    3:
	   HMI_AxisView[47].MoveReal:=FALSE;
       DO_[31,6].ON:=TRUE;
	   iAutoCut:=4;	
    4:
       tonAutoCut(IN:= TRUE, PT:= T#2S, Q=> , ET=> ); 
	   IF tonAutoCut.Q THEN 
	       tonAutoCut(IN:= FALSE, PT:= T#2S, Q=> , ET=> ); 
           iAutoCut:=5;	   
	   END_IF	
	   
    5: DO_[31,6].ON:=FALSE;
	   iAutoCut:=6;	
    6: 	  
       tonAutoCut(IN:= TRUE, PT:= T#3S, Q=> , ET=> ); 
	   IF tonAutoCut.Q THEN 
	       tonAutoCut(IN:= FALSE, PT:= T#3S, Q=> , ET=> ); 
           iAutoCut:=7;	   
	   END_IF	
    7: 
 	   IF icutcnt> HMI_cutCnt THEN
		  iAutoCut:=8; 
	   ELSE 
	      iAutoCut:=0; 
	   END_IF
	8:   
       HMI_AxisView[46].MoveReal:=TRUE;
	   iAutoCut:=9;	  
 
	9:
       tonAutoCut(IN:= TRUE, PT:= T#2S, Q=> , ET=> ); 
	   IF tonAutoCut.Q THEN 
	       tonAutoCut(IN:= FALSE, PT:= T#2S, Q=> , ET=> ); 
           iAutoCut:=10;	   
	   END_IF	
	   
	10:
	   icutcnt:=0;
       HMI_AxisView[46].MoveReal:=FALSE;
	   iAutoCut:=0;		   
	   
END_CASE


tonCounterAirOpen(IN:= glb_bCounterAirValve_UN01 , PT:= T#3S, Q=> , ET=> );
IF tonCounterAirOpen.Q THEN
   glb_bPackAirValve_UN01:=TRUE;
END_IF


IF HMI_DisableCntAlarmAll THEN
	FOR  i:=1 TO 40 DO
		HMI_SkipCntAlarm[i]:=TRUE;
	END_FOR
END_IF

IF HMI_EnbaleCntAlarmAll THEN
	FOR  i:=1 TO 40 DO
		HMI_SkipCntAlarm[i]:=FALSE;
	END_FOR	
END_IF

IF HMI_DisableCntAlarmAll2 THEN
	FOR  i:=1 TO 40 DO
		HMI_CntCheck[i]:=TRUE;
	END_FOR
END_IF

IF HMI_EnbaleCntAlarmAll2 THEN
	FOR  i:=1 TO 40 DO
		HMI_CntCheck[i]:=FALSE;
	END_FOR	
END_IF
END_ACTION

ACTION SR90_SafetyReset:
CASE iSafetyResetSeq OF
	0: IF glb_bSafetyReset THEN
		  iSafetyResetSeq:=10;
	   END_IF
	10: 	
		IF glb_arSafeRelayNo_UN01[1] OR tonSafetyReset.Q  THEN
		    iSafetyResetSeq:=20;
		END_IF
	20:	
		FOR i:=1 TO 64 DO
		    arRealAxisAdmin[i].i.Reset:= TRUE ;
			iSafetyResetSeq:=30;
		END_FOR		
	30:
	    IF tonSafetyReset.Q THEN
		   FOR i:=1 TO 64 DO
		       arRealAxisAdmin[i].i.Reset:= FALSE ;	
	       END_FOR	
		   glb_bSafetyreset:=FALSE;
		   iSafetyResetSeq:=0;
		END_IF
	
END_CASE

tonSafetyReset(IN:=glb_bSafetyreset , PT:=T#3S , Q=> , ET=> );

	
IF glb_arSafeRelayNo_UN01[1] THEN
	glb_bAllSafetyOk:=TRUE;
	ELSE 
	glb_bAllSafetyOk:=FALSE;
END_IF
END_ACTION

ACTION SR91_OEE:
HMI_OEEView.Active:=TRUE;
IF HMI_OEEView.Active THEN
   IF rtGoodCount.Q THEN	
      HMI_OEEView.GoodCount:= HMI_OEEView.GoodCount+7;	
   END_IF 
   IF rtNoGoodCount.Q THEN
	  HMI_OEEView.NoGoodCount:= HMI_OEEView.NoGoodCount+7;
   END_IF
  
END_IF

rtGoodCount(CLK:= glb_digoodFlag_UN01.11, Q=> );
rtNoGoodCount(CLK:= glb_diNogoodFlag_UN01.11 , Q=> );

IF HMI_OEEView.Reset THEN
   HMI_OEEView.GoodCount:=0;
   HMI_OEEView.NoGoodCount:=0;	
END_IF


HMI_OEEView.DesignSpeed:= 7.5;
HMI_OEEView.Performance:=HMI_OEEView.AverageSpeed/HMI_OEEView.DesignSpeed*100;


aoiActiveTotalTime(
	bEnable:= HMI_OEEView.Active, 
	bReset:= HMI_OEEView.Reset, 
	diSecond=> , 
	diMinute=> , 
	diHour=> , 
	diTotalSecond=> , 
	diTotalMinute=> HMI_OEEView.PlannedTime, 
	diTotalHour=> );

aoiWorkTotalTime(
	bEnable:= HMI_OEEView.Active AND Ref_MachineStateModel.Sts_Execute, 
	bReset:= HMI_OEEView.Reset, 
	diSecond=> , 
	diMinute=> , 
	diHour=> , 
	diTotalSecond=> , 
	diTotalMinute=> HMI_OEEView.UsableTime, 
	diTotalHour=> );

aoi10MinuteTime(
	bEnable:= bEn10Minute OR TRUE, 
	bReset:= bReset10Minute, 
	diSecond=> , 
	diMinute=> , 
	diHour=> , 
	diTotalSecond=> , 
	diTotalMinute=> , 
	diTotalHour=> );
	

HMI_OEEView.AverageSpeed:=DINT_TO_REAL(glb_TransferCnt)*7/DINT_TO_REAL(aoiWorkTotalTime.diTotalMinute);

	
IF	aoiActiveTotalTime.diTotalMinute>0 THEN
    HMI_OEEView.Usability:= DINT_TO_REAL(aoiWorkTotalTime.diTotalMinute)/DINT_TO_REAL(aoiActiveTotalTime.diTotalMinute)*100;
ELSE
    HMI_OEEView.Usability:= 0;
END_IF	

IF (HMI_OEEView.NoGoodCount+HMI_OEEView.GoodCount)> 0 THEN
    HMI_OEEView.Quality:=DINT_TO_REAL(HMI_OEEView.GoodCount)/(DINT_TO_REAL(HMI_OEEView.NoGoodCount)+DINT_TO_REAL(HMI_OEEView.GoodCount))*100;
ELSE
	HMI_OEEView.Quality:=0;
END_IF

HMI_OEEView.OEE:=(HMI_OEEView.Quality/100*HMI_OEEView.Usability/100*HMI_OEEView.Performance/100)*100;
END_ACTION

ACTION SR99_FaultClear:
CASE iFaultClearSeq OF
	0: 
		IF bClearAllFault THEN
		   iFaultClearSeq:=10;
		END_IF
	   
	10: 	
	//    IF NOT glb_bAirFeedback_UN01[2] THEN
	//		glb_bCounterAirValve_UN01:=FALSE;
	//	END_IF
	
	//	IF NOT glb_bAirFeedback_UN01[1] THEN
	//		glb_bPackAirValve_UN01:=FALSE;
	//	END_IF
		
		glb_MembraneAlarm:=FALSE;
		FOR i:=1 TO 50 DO
			IF arRealAxisAdmin[i].o.Error  THEN
			   arRealAxisAdmin[i].i.Reset:= TRUE ;
			END_IF
			IF arVirtualAxisAdmin[i].o.Error THEN
			   arVirtualAxisAdmin[i].i.Reset:= TRUE ;
			END_IF
		END_FOR
	
		FOR j:=1 TO 40 DO
			IF arDropCylinder[j].o.Error THEN
		       arDropCylinder[j].i.Reset:=TRUE;
			END_IF
			IF arCounters[j].Error THEN
			   arCounters[j].Clear:=TRUE;
			END_IF
		END_FOR
	    FOR j:=1 TO 50 DO
 			IF arPackCylinder[j].o.Error THEN
		       arPackCylinder[j].i.Reset:=TRUE;
			END_IF
			IF arPackVacuum[j].o.Error THEN
		       arPackVacuum[j].i.Reset:=TRUE;
			END_IF  
		END_FOR		
		
		FOR j:=1 TO 8 DO
			arHeat_AOI[j].Reset:=TRUE;
		END_FOR
        arDropBufferCyclinder[1].i.Reset:=TRUE;
		arDropBufferCyclinder[2].i.Reset:=TRUE;
	    iFaultClearSeq:=20;

	20:
		HMI_StopEvent[5].ID[20]:=FALSE;
		HMI_StopEvent[5].ID[21]:=FALSE;
		HMI_StopEvent[5].ID[22]:=FALSE;
		HMI_StopEvent[5].ID[23]:=FALSE;
		HMI_StopEvent[5].ID[24]:=FALSE;
		HMI_StopEvent[5].ID[25]:=FALSE;
		HMI_StopEvent[5].ID[26]:=FALSE;
	
	   IF  tonFaultClear.Q THEN 
			FOR i:=1 TO 50 DO
				 arRealAxisAdmin[i].i.Reset:= FALSE ;
				 arVirtualAxisAdmin[i].i.Reset:= FALSE ;
			END_FOR
			FOR j:=1 TO 40 DO
				arDropCylinder[j].i.Reset:=FALSE;
			    arCounters[j].Clear:=FALSE;				
			END_FOR
			FOR j:=1 TO 50 DO
				arPackCylinder[j].i.Reset:=FALSE;
				arPackVacuum[j].i.Reset:=FALSE;
			END_FOR			
			
			FOR j:=1 TO 8 DO
				arHeat_AOI[j].Reset:=FALSE;
			END_FOR
		    HMI_PrinterFault:=FALSE;
			
		    HMI_StopEvent[0].ID[6]:=FALSE;
		    HMI_StopEvent[0].ID[7]:=FALSE;
			
		//	glb_bPackAirValve_UN01:=TRUE;
		//	glb_bCounterAirValve_UN01:=TRUE;
		
		    arDropBufferCyclinder[1].i.Reset:=FALSE;
		    arDropBufferCyclinder[2].i.Reset:=FALSE;
		
			HMI_AlarmMute:=FALSE;
			bClearAllFault:=FALSE;
			iFaultClearSeq:=0;
       END_IF
	   
END_CASE

tonFaultClear(IN:=bClearAllFault , PT:=T#500MS , Q=> , ET=> );
END_ACTION

ACTION UP01_PackML:
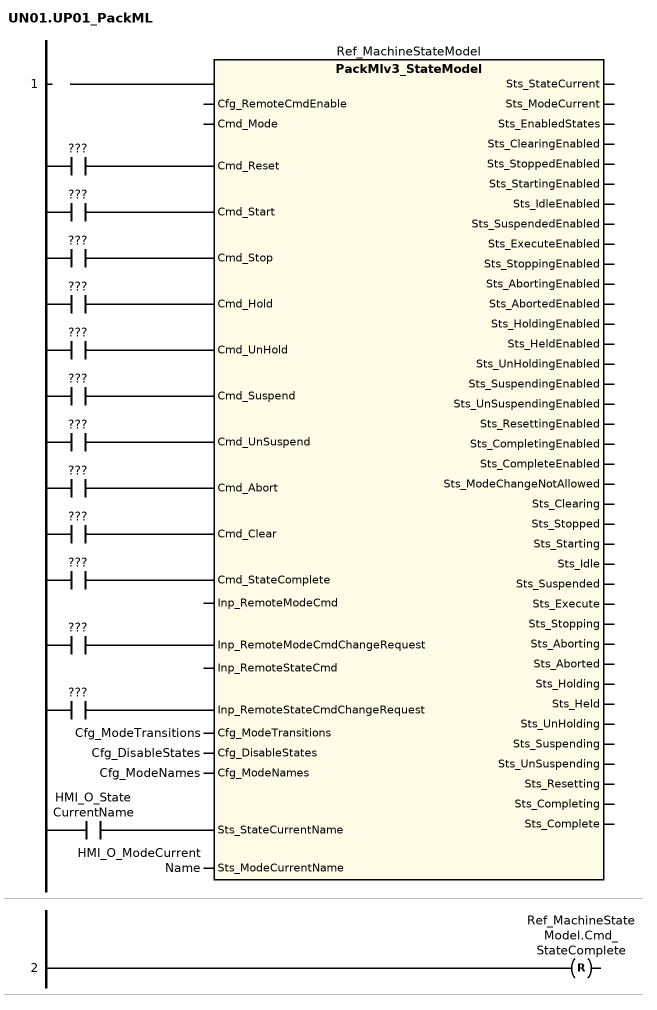
// NETWORK 1
Ref_MachineStateModel(
    Cfg_ModeTransitions := Cfg_ModeTransitions,
    Cfg_DisableStates := Cfg_DisableStates,
    Cfg_ModeNames := Cfg_ModeNames,
    Sts_StateCurrentName := HMI_O_StateCurrentName,
    Sts_ModeCurrentName := HMI_O_ModeCurrentName); // PackMlv3_StateModel

// NETWORK 2
Ref_MachineStateModel.Cmd_StateComplete R= TRUE;
END_ACTION

ACTION UP02_StateComplete:
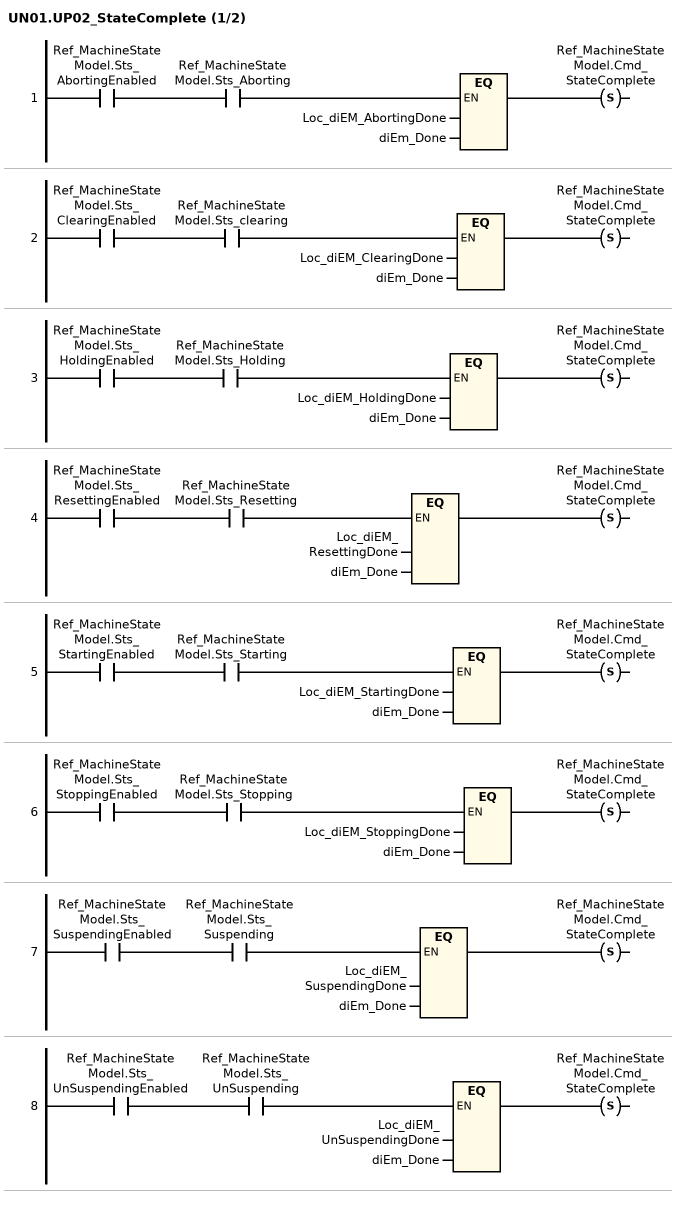
// NETWORK 1
Ref_MachineStateModel.Cmd_StateComplete S= Ref_MachineStateModel.Sts_AbortingEnabled AND Ref_MachineStateModel.Sts_Aborting AND Loc_diEM_AbortingDone = diEm_Done;

// NETWORK 2
Ref_MachineStateModel.Cmd_StateComplete S= Ref_MachineStateModel.Sts_ClearingEnabled AND Ref_MachineStateModel.Sts_clearing AND Loc_diEM_ClearingDone = diEm_Done;

// NETWORK 3
Ref_MachineStateModel.Cmd_StateComplete S= Ref_MachineStateModel.Sts_HoldingEnabled AND Ref_MachineStateModel.Sts_Holding AND Loc_diEM_HoldingDone = diEm_Done;

// NETWORK 4
Ref_MachineStateModel.Cmd_StateComplete S= Ref_MachineStateModel.Sts_ResettingEnabled AND Ref_MachineStateModel.Sts_Resetting AND Loc_diEM_ResettingDone = diEm_Done;

// NETWORK 5
Ref_MachineStateModel.Cmd_StateComplete S= Ref_MachineStateModel.Sts_StartingEnabled AND Ref_MachineStateModel.Sts_Starting AND Loc_diEM_StartingDone = diEm_Done;

// NETWORK 6
Ref_MachineStateModel.Cmd_StateComplete S= Ref_MachineStateModel.Sts_StoppingEnabled AND Ref_MachineStateModel.Sts_Stopping AND Loc_diEM_StoppingDone = diEm_Done;

// NETWORK 7
Ref_MachineStateModel.Cmd_StateComplete S= Ref_MachineStateModel.Sts_SuspendingEnabled AND Ref_MachineStateModel.Sts_Suspending AND Loc_diEM_SuspendingDone = diEm_Done;

// NETWORK 8
Ref_MachineStateModel.Cmd_StateComplete S= Ref_MachineStateModel.Sts_UnSuspendingEnabled AND Ref_MachineStateModel.Sts_UnSuspending AND Loc_diEM_UnSuspendingDone = diEm_Done;

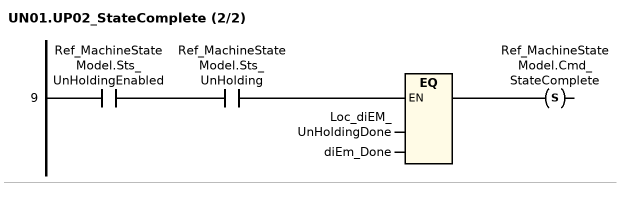
// NETWORK 9
Ref_MachineStateModel.Cmd_StateComplete S= Ref_MachineStateModel.Sts_UnHoldingEnabled AND Ref_MachineStateModel.Sts_UnHolding AND Loc_diEM_UnHoldingDone = diEm_Done;
END_ACTION

END_PROGRAM

// ---- Add-On-Instructions/PackMlv3_StateModel.TcPOU
FUNCTION_BLOCK PackMlv3_StateModel
VAR_INPUT
	Cfg_RemoteCmdEnable: BOOL;
	Cmd_Mode: DINT;
	Cmd_Reset: BOOL;
	Cmd_Start: BOOL;
	Cmd_Stop: BOOL;
	Cmd_Hold: BOOL;
	Cmd_UnHold: BOOL;
	Cmd_Suspend: BOOL;
	Cmd_UnSuspend: BOOL;
	Cmd_Abort: BOOL;
	Cmd_Clear: BOOL;
	Cmd_StateComplete: BOOL;
	Inp_RemoteModeCmd: DINT;
	Inp_RemoteModeCmdChangeRequest: BOOL;
	Inp_RemoteStateCmd: DINT;
	Inp_RemoteStateCmdChangeRequest: BOOL;
END_VAR
VAR_OUTPUT
	Sts_StateCurrent: DINT;
	Sts_ModeCurrent: DINT;
	Sts_EnabledStates: DINT;
	Sts_ClearingEnabled: BOOL;
	Sts_StoppedEnabled: BOOL;
	Sts_StartingEnabled: BOOL;
	Sts_IdleEnabled: BOOL;
	Sts_SuspendedEnabled: BOOL;
	Sts_ExecuteEnabled: BOOL;
	Sts_StoppingEnabled: BOOL;
	Sts_AbortingEnabled: BOOL;
	Sts_AbortedEnabled: BOOL;
	Sts_HoldingEnabled: BOOL;
	Sts_HeldEnabled: BOOL;
	Sts_UnHoldingEnabled: BOOL;
	Sts_SuspendingEnabled: BOOL;
	Sts_UnSuspendingEnabled: BOOL;
	Sts_ResettingEnabled: BOOL;
	Sts_CompletingEnabled: BOOL;
	Sts_CompleteEnabled: BOOL;
	Sts_ModeChangeNotAllowed: BOOL;
	Sts_Clearing: BOOL;
	Sts_Stopped: BOOL;
	Sts_Starting: BOOL;
	Sts_Idle: BOOL;
	Sts_Suspended: BOOL;
	Sts_Execute: BOOL;
	Sts_Stopping: BOOL;
	Sts_Aborting: BOOL;
	Sts_Aborted: BOOL;
	Sts_Holding: BOOL;
	Sts_Held: BOOL;
	Sts_UnHolding: BOOL;
	Sts_Suspending: BOOL;
	Sts_UnSuspending: BOOL;
	Sts_Resetting: BOOL;
	Sts_Completing: BOOL;
	Sts_Complete: BOOL;
END_VAR
VAR_IN_OUT
	Cfg_ModeTransitions: ARRAY[0..31] OF DINT;
	Cfg_DisableStates: ARRAY[0..31] OF DINT;
	Cfg_ModeNames: ARRAY[0..31] OF STRING;
	Sts_StateCurrentName: STRING(255);	
	Sts_ModeCurrentName: STRING(255);	
END_VAR
VAR
	RemoteCmdChangeRequested: BOOL;
	ResetRemoteCmd: BOOL;
	StartRemoteCmd: BOOL;
	StopRemoteCmd: BOOL;
	HoldRemoteCmd: BOOL;
	UnholdRemoteCmd: BOOL;
	SuspendRemoteCmd: BOOL;
	UnSuspendRemoteCmd: BOOL;
	AbortRemoteCmd: BOOL;
	ClearRemoteCmd: BOOL;
	Cfg_DisableStatesCopy: DINT;
	StateComplete: BOOL;
	LocalClearing: BOOL;
	LocalStopped: BOOL;
	LocalStarting: BOOL;
	LocalExecute: BOOL;
	LocalCompleting: BOOL;
	LocalStopping: BOOL;
	LocalAborting: BOOL;
	LocalAborted: BOOL;
	LocalHolding: BOOL;
	LocalHeld: BOOL;
	LocalUnHolding: BOOL;
	LocalSuspending: BOOL;
	LocalSuspended: BOOL;
	LocalUnSuspending: BOOL;
	LocalResetting: BOOL;
	LocalIdle: BOOL;
	LocalComplete: BOOL;
	END_IFIF: INT;
	FS: BOOL;
END_VAR
VAR // added by the converter: edge detectors and wires of the graphical bodies
    _w1, _w2, _w3, _w4, _w5, _w6, _w7, _w8, _w9, _w10, _w11, _w12, _w13, _w14, _w15, _w16, _w17, _w18, _w19, _w20, _w21, _w22, _w23, _w24, _w25, _w26, _w27, _w28, _w29, _w30, _w31, _w32, _w33, _w34, _w35, _w36, _w37, _w38, _w39, _w40, _w41, _w42, _w43, _w44, _w45, _w46, _w47, _w48, _w49, _w50, _w51, _w52, _w53, _w54, _w55, _w56 : BOOL;
END_VAR


IF NOT FS THEN
	Sts_ModeCurrent:=1;
	Cmd_Mode:=1;
	StS_StateCurrent:=2;
    LocalClearing:=FALSE;
	LocalStopped:=TRUE;
	LocalStarting:=FALSE;
	LocalExecute:=FALSE;
	LocalCompleting:=FALSE;
	LocalStopping:=FALSE;
	LocalAborting:=FALSE;
	LocalAborted:=FALSE;
	LocalHolding:=FALSE;
	LocalHeld:=FALSE;
	LocalUnHolding:=FALSE;
	LocalSuspending:=FALSE;
	LocalSuspended:=FALSE;
	LocalUnSuspending:=FALSE;
	LocalResetting:=FALSE;
	LocalIdle:=FALSE;
	LocalComplete:=FALSE;
	FS:=TRUE;
END_IF
ACT();

IF Sts_StateCurrent=0 THEN
	IF RemoteCmdchangerequested AND inp_remoteModeCmd<>0 AND Inp_RemoteModeCmd>1 AND Inp_RemoteModeCmd<32 
	 AND Cfg_ModeTransitions[Sts_ModeCurrent].0 AND Cfg_ModeTransitions[Inp_RemoteModeCmd].0 THEN
		Sts_ModeCurrent:=Inp_RemoteModeCmd;
		Cmd_Mode:=Sts_ModeCurrent;
	END_IF
	IF Cmd_Mode<>Sts_ModeCurrent AND Cmd_Mode>1 AND Cmd_Mode<32 
	 AND Cfg_ModeTransitions[Sts_ModeCurrent].0 AND Cfg_ModeTransitions[Cmd_Mode].0 THEN	
		Sts_ModeCurrent:=Cmd_Mode;
	END_IF
	
END_IF
IF Sts_StateCurrent=1 THEN
	IF RemoteCmdchangerequested AND inp_remoteModeCmd<>0 AND Inp_RemoteModeCmd>1 AND Inp_RemoteModeCmd<32 
	 AND Cfg_ModeTransitions[Sts_ModeCurrent].1 AND Cfg_ModeTransitions[Inp_RemoteModeCmd].1 THEN
		Sts_ModeCurrent:=Inp_RemoteModeCmd;
		Cmd_Mode:=Sts_ModeCurrent;
	END_IF
	IF Cmd_Mode<>Sts_ModeCurrent AND Cmd_Mode>1 AND Cmd_Mode<32 
	 AND Cfg_ModeTransitions[Sts_ModeCurrent].1 AND Cfg_ModeTransitions[Cmd_Mode].1 THEN	
		Sts_ModeCurrent:=Cmd_Mode;
	END_IF
END_IF
IF Sts_StateCurrent=2 THEN
	IF RemoteCmdchangerequested AND inp_remoteModeCmd<>0 AND Inp_RemoteModeCmd>1 AND Inp_RemoteModeCmd<32 
	 AND Cfg_ModeTransitions[Sts_ModeCurrent].2 AND Cfg_ModeTransitions[Inp_RemoteModeCmd].2 THEN
		Sts_ModeCurrent:=Inp_RemoteModeCmd;
		Cmd_Mode:=Sts_ModeCurrent;
	END_IF
	IF Cmd_Mode<>Sts_ModeCurrent AND Cmd_Mode>1 AND Cmd_Mode<32 
	 AND Cfg_ModeTransitions[Sts_ModeCurrent].2 AND Cfg_ModeTransitions[Cmd_Mode].2 THEN	
		Sts_ModeCurrent:=Cmd_Mode;
	END_IF
END_IF
IF Sts_StateCurrent=3 THEN
	IF RemoteCmdchangerequested AND inp_remoteModeCmd<>0 AND Inp_RemoteModeCmd>1 AND Inp_RemoteModeCmd<32 
	 AND Cfg_ModeTransitions[Sts_ModeCurrent].3 AND Cfg_ModeTransitions[Inp_RemoteModeCmd].3 THEN
		Sts_ModeCurrent:=Inp_RemoteModeCmd;
		Cmd_Mode:=Sts_ModeCurrent;
	END_IF
	IF Cmd_Mode<>Sts_ModeCurrent AND Cmd_Mode>1 AND Cmd_Mode<32 
	 AND Cfg_ModeTransitions[Sts_ModeCurrent].3 AND Cfg_ModeTransitions[Cmd_Mode].3 THEN	
		Sts_ModeCurrent:=Cmd_Mode;
	END_IF
END_IF
IF Sts_StateCurrent=4 THEN
	IF RemoteCmdchangerequested AND inp_remoteModeCmd<>0 AND Inp_RemoteModeCmd>1 AND Inp_RemoteModeCmd<32 
	 AND Cfg_ModeTransitions[Sts_ModeCurrent].4 AND Cfg_ModeTransitions[Inp_RemoteModeCmd].4 THEN
		Sts_ModeCurrent:=Inp_RemoteModeCmd;
		Cmd_Mode:=Sts_ModeCurrent;
	END_IF
	IF Cmd_Mode<>Sts_ModeCurrent AND Cmd_Mode>1 AND Cmd_Mode<32 
	 AND Cfg_ModeTransitions[Sts_ModeCurrent].4 AND Cfg_ModeTransitions[Cmd_Mode].4 THEN	
		Sts_ModeCurrent:=Cmd_Mode;
	END_IF
END_IF
IF Sts_StateCurrent=5 THEN
	IF RemoteCmdchangerequested AND inp_remoteModeCmd<>0 AND Inp_RemoteModeCmd>1 AND Inp_RemoteModeCmd<32 
	 AND Cfg_ModeTransitions[Sts_ModeCurrent].5 AND Cfg_ModeTransitions[Inp_RemoteModeCmd].5 THEN
		Sts_ModeCurrent:=Inp_RemoteModeCmd;
		Cmd_Mode:=Sts_ModeCurrent;
	END_IF
	IF Cmd_Mode<>Sts_ModeCurrent AND Cmd_Mode>1 AND Cmd_Mode<32 
	 AND Cfg_ModeTransitions[Sts_ModeCurrent].5 AND Cfg_ModeTransitions[Cmd_Mode].5 THEN	
		Sts_ModeCurrent:=Cmd_Mode;
	END_IF
END_IF
IF Sts_StateCurrent=6 THEN
	IF RemoteCmdchangerequested AND inp_remoteModeCmd<>0 AND Inp_RemoteModeCmd>1 AND Inp_RemoteModeCmd<32 
	 AND Cfg_ModeTransitions[Sts_ModeCurrent].6 AND Cfg_ModeTransitions[Inp_RemoteModeCmd].6 THEN
		Sts_ModeCurrent:=Inp_RemoteModeCmd;
		Cmd_Mode:=Sts_ModeCurrent;
	END_IF
	IF Cmd_Mode<>Sts_ModeCurrent AND Cmd_Mode>1 AND Cmd_Mode<32 
	 AND Cfg_ModeTransitions[Sts_ModeCurrent].6 AND Cfg_ModeTransitions[Cmd_Mode].6 THEN	
		Sts_ModeCurrent:=Cmd_Mode;
	END_IF
END_IF
IF Sts_StateCurrent=7 THEN
	IF RemoteCmdchangerequested AND inp_remoteModeCmd<>0 AND Inp_RemoteModeCmd>1 AND Inp_RemoteModeCmd<32 
	 AND Cfg_ModeTransitions[Sts_ModeCurrent].7 AND Cfg_ModeTransitions[Inp_RemoteModeCmd].7 THEN
		Sts_ModeCurrent:=Inp_RemoteModeCmd;
		Cmd_Mode:=Sts_ModeCurrent;
	END_IF
	IF Cmd_Mode<>Sts_ModeCurrent AND Cmd_Mode>1 AND Cmd_Mode<32 
	 AND Cfg_ModeTransitions[Sts_ModeCurrent].7 AND Cfg_ModeTransitions[Cmd_Mode].7 THEN	
		Sts_ModeCurrent:=Cmd_Mode;
	END_IF
END_IF
IF Sts_StateCurrent=8 THEN
	IF RemoteCmdchangerequested AND inp_remoteModeCmd<>0 AND Inp_RemoteModeCmd>1 AND Inp_RemoteModeCmd<32 
	 AND Cfg_ModeTransitions[Sts_ModeCurrent].8 AND Cfg_ModeTransitions[Inp_RemoteModeCmd].8 THEN
		Sts_ModeCurrent:=Inp_RemoteModeCmd;
		Cmd_Mode:=Sts_ModeCurrent;
	END_IF
	IF Cmd_Mode<>Sts_ModeCurrent AND Cmd_Mode>1 AND Cmd_Mode<32 
	 AND Cfg_ModeTransitions[Sts_ModeCurrent].8 AND Cfg_ModeTransitions[Cmd_Mode].8 THEN	
		Sts_ModeCurrent:=Cmd_Mode;
	END_IF
END_IF
IF Sts_StateCurrent=9 THEN
	IF RemoteCmdchangerequested AND inp_remoteModeCmd<>0 AND Inp_RemoteModeCmd>1 AND Inp_RemoteModeCmd<32 
	 AND Cfg_ModeTransitions[Sts_ModeCurrent].9 AND Cfg_ModeTransitions[Inp_RemoteModeCmd].9 THEN
		Sts_ModeCurrent:=Inp_RemoteModeCmd;
		Cmd_Mode:=Sts_ModeCurrent;
	END_IF
	IF Cmd_Mode<>Sts_ModeCurrent AND Cmd_Mode>1 AND Cmd_Mode<32 
	 AND Cfg_ModeTransitions[Sts_ModeCurrent].9 AND Cfg_ModeTransitions[Cmd_Mode].9 THEN	
		Sts_ModeCurrent:=Cmd_Mode;
	END_IF
END_IF
IF Sts_StateCurrent=10 THEN
	IF RemoteCmdchangerequested AND inp_remoteModeCmd<>0 AND Inp_RemoteModeCmd>1 AND Inp_RemoteModeCmd<32 
	 AND Cfg_ModeTransitions[Sts_ModeCurrent].10 AND Cfg_ModeTransitions[Inp_RemoteModeCmd].10 THEN
		Sts_ModeCurrent:=Inp_RemoteModeCmd;
		Cmd_Mode:=Sts_ModeCurrent;
	END_IF
	IF Cmd_Mode<>Sts_ModeCurrent AND Cmd_Mode>1 AND Cmd_Mode<32 
	 AND Cfg_ModeTransitions[Sts_ModeCurrent].10 AND Cfg_ModeTransitions[Cmd_Mode].10 THEN	
		Sts_ModeCurrent:=Cmd_Mode;
	END_IF
END_IF
IF Sts_StateCurrent=11 THEN
	IF RemoteCmdchangerequested AND inp_remoteModeCmd<>0 AND Inp_RemoteModeCmd>1 AND Inp_RemoteModeCmd<32 
	 AND Cfg_ModeTransitions[Sts_ModeCurrent].11 AND Cfg_ModeTransitions[Inp_RemoteModeCmd].11 THEN
		Sts_ModeCurrent:=Inp_RemoteModeCmd;
		Cmd_Mode:=Sts_ModeCurrent;
	END_IF
	IF Cmd_Mode<>Sts_ModeCurrent AND Cmd_Mode>1 AND Cmd_Mode<32 
	 AND Cfg_ModeTransitions[Sts_ModeCurrent].11 AND Cfg_ModeTransitions[Cmd_Mode].11 THEN	
		Sts_ModeCurrent:=Cmd_Mode;
	END_IF
END_IF
IF Sts_StateCurrent=12 THEN
	IF RemoteCmdchangerequested AND inp_remoteModeCmd<>0 AND Inp_RemoteModeCmd>1 AND Inp_RemoteModeCmd<32 
	 AND Cfg_ModeTransitions[Sts_ModeCurrent].12 AND Cfg_ModeTransitions[Inp_RemoteModeCmd].12 THEN
		Sts_ModeCurrent:=Inp_RemoteModeCmd;
		Cmd_Mode:=Sts_ModeCurrent;
	END_IF
	IF Cmd_Mode<>Sts_ModeCurrent AND Cmd_Mode>1 AND Cmd_Mode<32 
	 AND Cfg_ModeTransitions[Sts_ModeCurrent].12 AND Cfg_ModeTransitions[Cmd_Mode].12 THEN	
		Sts_ModeCurrent:=Cmd_Mode;
	END_IF
END_IF
IF Sts_StateCurrent=13 THEN
	IF RemoteCmdchangerequested AND inp_remoteModeCmd<>0 AND Inp_RemoteModeCmd>1 AND Inp_RemoteModeCmd<32 
	 AND Cfg_ModeTransitions[Sts_ModeCurrent].13 AND Cfg_ModeTransitions[Inp_RemoteModeCmd].13 THEN
		Sts_ModeCurrent:=Inp_RemoteModeCmd;
		Cmd_Mode:=Sts_ModeCurrent;
	END_IF
	IF Cmd_Mode<>Sts_ModeCurrent AND Cmd_Mode>1 AND Cmd_Mode<32 
	 AND Cfg_ModeTransitions[Sts_ModeCurrent].13 AND Cfg_ModeTransitions[Cmd_Mode].13 THEN	
		Sts_ModeCurrent:=Cmd_Mode;
	END_IF
END_IF
IF Sts_StateCurrent=14 THEN
	IF RemoteCmdchangerequested AND inp_remoteModeCmd<>0 AND Inp_RemoteModeCmd>1 AND Inp_RemoteModeCmd<32 
	 AND Cfg_ModeTransitions[Sts_ModeCurrent].14 AND Cfg_ModeTransitions[Inp_RemoteModeCmd].14 THEN
		Sts_ModeCurrent:=Inp_RemoteModeCmd;
		Cmd_Mode:=Sts_ModeCurrent;
	END_IF
	IF Cmd_Mode<>Sts_ModeCurrent AND Cmd_Mode>1 AND Cmd_Mode<32 
	 AND Cfg_ModeTransitions[Sts_ModeCurrent].14 AND Cfg_ModeTransitions[Cmd_Mode].14 THEN	
		Sts_ModeCurrent:=Cmd_Mode;
	END_IF
END_IF
IF Sts_StateCurrent=15 THEN
	IF RemoteCmdchangerequested AND inp_remoteModeCmd<>0 AND Inp_RemoteModeCmd>1 AND Inp_RemoteModeCmd<32 
	 AND Cfg_ModeTransitions[Sts_ModeCurrent].15 AND Cfg_ModeTransitions[Inp_RemoteModeCmd].15 THEN
		Sts_ModeCurrent:=Inp_RemoteModeCmd;
		Cmd_Mode:=Sts_ModeCurrent;
	END_IF
	IF Cmd_Mode<>Sts_ModeCurrent AND Cmd_Mode>1 AND Cmd_Mode<32 
	 AND Cfg_ModeTransitions[Sts_ModeCurrent].15 AND Cfg_ModeTransitions[Cmd_Mode].15 THEN	
		Sts_ModeCurrent:=Cmd_Mode;
	END_IF
END_IF
IF Sts_StateCurrent=16 THEN
	IF RemoteCmdchangerequested AND inp_remoteModeCmd<>0 AND Inp_RemoteModeCmd>1 AND Inp_RemoteModeCmd<32 
	 AND Cfg_ModeTransitions[Sts_ModeCurrent].16 AND Cfg_ModeTransitions[Inp_RemoteModeCmd].16 THEN
		Sts_ModeCurrent:=Inp_RemoteModeCmd;
		Cmd_Mode:=Sts_ModeCurrent;
	END_IF
	IF Cmd_Mode<>Sts_ModeCurrent AND Cmd_Mode>1 AND Cmd_Mode<32 
	 AND Cfg_ModeTransitions[Sts_ModeCurrent].16 AND Cfg_ModeTransitions[Cmd_Mode].16 THEN	
		Sts_ModeCurrent:=Cmd_Mode;
	END_IF
END_IF	
IF Sts_StateCurrent=17 THEN
	IF RemoteCmdchangerequested AND inp_remoteModeCmd<>0 AND Inp_RemoteModeCmd>1 AND Inp_RemoteModeCmd<32 
	 AND Cfg_ModeTransitions[Sts_ModeCurrent].17 AND Cfg_ModeTransitions[Inp_RemoteModeCmd].17 THEN
		Sts_ModeCurrent:=Inp_RemoteModeCmd;
		Cmd_Mode:=Sts_ModeCurrent;
	END_IF
	IF Cmd_Mode<>Sts_ModeCurrent AND Cmd_Mode>1 AND Cmd_Mode<32 
	 AND Cfg_ModeTransitions[Sts_ModeCurrent].17 AND Cfg_ModeTransitions[Cmd_Mode].17 THEN	
		Sts_ModeCurrent:=Cmd_Mode;
	END_IF
END_IF
IF Sts_StateCurrent=18 THEN
	IF RemoteCmdchangerequested AND inp_remoteModeCmd<>0 AND Inp_RemoteModeCmd>1 AND Inp_RemoteModeCmd<32 
	 AND Cfg_ModeTransitions[Sts_ModeCurrent].18 AND Cfg_ModeTransitions[Inp_RemoteModeCmd].18 THEN
		Sts_ModeCurrent:=Inp_RemoteModeCmd;
		Cmd_Mode:=Sts_ModeCurrent;
	END_IF
	IF Cmd_Mode<>Sts_ModeCurrent AND Cmd_Mode>1 AND Cmd_Mode<32 
	 AND Cfg_ModeTransitions[Sts_ModeCurrent].18 AND Cfg_ModeTransitions[Cmd_Mode].18 THEN	
		Sts_ModeCurrent:=Cmd_Mode;
	END_IF
END_IF
IF Sts_StateCurrent=19 THEN
	IF RemoteCmdchangerequested AND inp_remoteModeCmd<>0 AND Inp_RemoteModeCmd>1 AND Inp_RemoteModeCmd<32 
	 AND Cfg_ModeTransitions[Sts_ModeCurrent].19 AND Cfg_ModeTransitions[Inp_RemoteModeCmd].19 THEN
		Sts_ModeCurrent:=Inp_RemoteModeCmd;
		Cmd_Mode:=Sts_ModeCurrent;
	END_IF
	IF Cmd_Mode<>Sts_ModeCurrent AND Cmd_Mode>1 AND Cmd_Mode<32 
	 AND Cfg_ModeTransitions[Sts_ModeCurrent].19 AND Cfg_ModeTransitions[Cmd_Mode].19 THEN	
		Sts_ModeCurrent:=Cmd_Mode;
	END_IF
END_IF
IF Sts_StateCurrent=20 THEN
	IF RemoteCmdchangerequested AND inp_remoteModeCmd<>0 AND Inp_RemoteModeCmd>1 AND Inp_RemoteModeCmd<32 
	 AND Cfg_ModeTransitions[Sts_ModeCurrent].20 AND Cfg_ModeTransitions[Inp_RemoteModeCmd].20 THEN
		Sts_ModeCurrent:=Inp_RemoteModeCmd;
		Cmd_Mode:=Sts_ModeCurrent;
	END_IF
	IF Cmd_Mode<>Sts_ModeCurrent AND Cmd_Mode>1 AND Cmd_Mode<32 
	 AND Cfg_ModeTransitions[Sts_ModeCurrent].20 AND Cfg_ModeTransitions[Cmd_Mode].20 THEN	
		Sts_ModeCurrent:=Cmd_Mode;
	END_IF
END_IF
IF Sts_StateCurrent=21 THEN
	IF RemoteCmdchangerequested AND inp_remoteModeCmd<>0 AND Inp_RemoteModeCmd>1 AND Inp_RemoteModeCmd<32 
	 AND Cfg_ModeTransitions[Sts_ModeCurrent].21 AND Cfg_ModeTransitions[Inp_RemoteModeCmd].21 THEN
		Sts_ModeCurrent:=Inp_RemoteModeCmd;
		Cmd_Mode:=Sts_ModeCurrent;
	END_IF
	IF Cmd_Mode<>Sts_ModeCurrent AND Cmd_Mode>1 AND Cmd_Mode<32 
	 AND Cfg_ModeTransitions[Sts_ModeCurrent].21 AND Cfg_ModeTransitions[Cmd_Mode].21 THEN	
		Sts_ModeCurrent:=Cmd_Mode;
	END_IF
END_IF
IF Sts_StateCurrent=22 THEN
	IF RemoteCmdchangerequested AND inp_remoteModeCmd<>0 AND Inp_RemoteModeCmd>1 AND Inp_RemoteModeCmd<32 
	 AND Cfg_ModeTransitions[Sts_ModeCurrent].22 AND Cfg_ModeTransitions[Inp_RemoteModeCmd].22 THEN
		Sts_ModeCurrent:=Inp_RemoteModeCmd;
		Cmd_Mode:=Sts_ModeCurrent;
	END_IF
	IF Cmd_Mode<>Sts_ModeCurrent AND Cmd_Mode>1 AND Cmd_Mode<32 
	 AND Cfg_ModeTransitions[Sts_ModeCurrent].22 AND Cfg_ModeTransitions[Cmd_Mode].22 THEN	
		Sts_ModeCurrent:=Cmd_Mode;
	END_IF
END_IF
IF Sts_StateCurrent=23 THEN
	IF RemoteCmdchangerequested AND inp_remoteModeCmd<>0 AND Inp_RemoteModeCmd>1 AND Inp_RemoteModeCmd<32 
	 AND Cfg_ModeTransitions[Sts_ModeCurrent].23 AND Cfg_ModeTransitions[Inp_RemoteModeCmd].23 THEN
		Sts_ModeCurrent:=Inp_RemoteModeCmd;
		Cmd_Mode:=Sts_ModeCurrent;
	END_IF
	IF Cmd_Mode<>Sts_ModeCurrent AND Cmd_Mode>1 AND Cmd_Mode<32 
	 AND Cfg_ModeTransitions[Sts_ModeCurrent].23 AND Cfg_ModeTransitions[Cmd_Mode].23 THEN	
		Sts_ModeCurrent:=Cmd_Mode;
	END_IF
END_IF
IF Sts_StateCurrent=24 THEN
	IF RemoteCmdchangerequested AND inp_remoteModeCmd<>0 AND Inp_RemoteModeCmd>1 AND Inp_RemoteModeCmd<32 
	 AND Cfg_ModeTransitions[Sts_ModeCurrent].24 AND Cfg_ModeTransitions[Inp_RemoteModeCmd].24 THEN
		Sts_ModeCurrent:=Inp_RemoteModeCmd;
		Cmd_Mode:=Sts_ModeCurrent;
	END_IF
	IF Cmd_Mode<>Sts_ModeCurrent AND Cmd_Mode>1 AND Cmd_Mode<32 
	 AND Cfg_ModeTransitions[Sts_ModeCurrent].24 AND Cfg_ModeTransitions[Cmd_Mode].24 THEN	
		Sts_ModeCurrent:=Cmd_Mode;
	END_IF
END_IF
IF Sts_StateCurrent=25 THEN
	IF RemoteCmdchangerequested AND inp_remoteModeCmd<>0 AND Inp_RemoteModeCmd>1 AND Inp_RemoteModeCmd<32 
	 AND Cfg_ModeTransitions[Sts_ModeCurrent].25 AND Cfg_ModeTransitions[Inp_RemoteModeCmd].25 THEN
		Sts_ModeCurrent:=Inp_RemoteModeCmd;
		Cmd_Mode:=Sts_ModeCurrent;
	END_IF
	IF Cmd_Mode<>Sts_ModeCurrent AND Cmd_Mode>1 AND Cmd_Mode<32 
	 AND Cfg_ModeTransitions[Sts_ModeCurrent].25 AND Cfg_ModeTransitions[Cmd_Mode].25 THEN	
		Sts_ModeCurrent:=Cmd_Mode;
	END_IF
END_IF
IF Sts_StateCurrent=26 THEN
	IF RemoteCmdchangerequested AND inp_remoteModeCmd<>0 AND Inp_RemoteModeCmd>1 AND Inp_RemoteModeCmd<32 
	 AND Cfg_ModeTransitions[Sts_ModeCurrent].26 AND Cfg_ModeTransitions[Inp_RemoteModeCmd].26 THEN
		Sts_ModeCurrent:=Inp_RemoteModeCmd;
		Cmd_Mode:=Sts_ModeCurrent;
	END_IF
	IF Cmd_Mode<>Sts_ModeCurrent AND Cmd_Mode>1 AND Cmd_Mode<32 
	 AND Cfg_ModeTransitions[Sts_ModeCurrent].26 AND Cfg_ModeTransitions[Cmd_Mode].26 THEN	
		Sts_ModeCurrent:=Cmd_Mode;
	END_IF
END_IF
IF Sts_StateCurrent=27 THEN
	IF RemoteCmdchangerequested AND inp_remoteModeCmd<>0 AND Inp_RemoteModeCmd>1 AND Inp_RemoteModeCmd<32 
	 AND Cfg_ModeTransitions[Sts_ModeCurrent].27 AND Cfg_ModeTransitions[Inp_RemoteModeCmd].27 THEN
		Sts_ModeCurrent:=Inp_RemoteModeCmd;
		Cmd_Mode:=Sts_ModeCurrent;
	END_IF
	IF Cmd_Mode<>Sts_ModeCurrent AND Cmd_Mode>1 AND Cmd_Mode<32 
	 AND Cfg_ModeTransitions[Sts_ModeCurrent].27 AND Cfg_ModeTransitions[Cmd_Mode].27 THEN	
		Sts_ModeCurrent:=Cmd_Mode;
	END_IF
END_IF
IF Sts_StateCurrent=28 THEN
	IF RemoteCmdchangerequested AND inp_remoteModeCmd<>0 AND Inp_RemoteModeCmd>1 AND Inp_RemoteModeCmd<32 
	 AND Cfg_ModeTransitions[Sts_ModeCurrent].28 AND Cfg_ModeTransitions[Inp_RemoteModeCmd].28 THEN
		Sts_ModeCurrent:=Inp_RemoteModeCmd;
		Cmd_Mode:=Sts_ModeCurrent;
	END_IF
	IF Cmd_Mode<>Sts_ModeCurrent AND Cmd_Mode>1 AND Cmd_Mode<32 
	 AND Cfg_ModeTransitions[Sts_ModeCurrent].28 AND Cfg_ModeTransitions[Cmd_Mode].28 THEN	
		Sts_ModeCurrent:=Cmd_Mode;
	END_IF
END_IF
IF Sts_StateCurrent=29 THEN
	IF RemoteCmdchangerequested AND inp_remoteModeCmd<>0 AND Inp_RemoteModeCmd>1 AND Inp_RemoteModeCmd<32 
	 AND Cfg_ModeTransitions[Sts_ModeCurrent].29 AND Cfg_ModeTransitions[Inp_RemoteModeCmd].29 THEN
		Sts_ModeCurrent:=Inp_RemoteModeCmd;
		Cmd_Mode:=Sts_ModeCurrent;
	END_IF
	IF Cmd_Mode<>Sts_ModeCurrent AND Cmd_Mode>1 AND Cmd_Mode<32 
	 AND Cfg_ModeTransitions[Sts_ModeCurrent].29 AND Cfg_ModeTransitions[Cmd_Mode].29 THEN	
		Sts_ModeCurrent:=Cmd_Mode;
	END_IF
END_IF
IF Sts_StateCurrent=30 THEN
	IF RemoteCmdchangerequested AND inp_remoteModeCmd<>0 AND Inp_RemoteModeCmd>1 AND Inp_RemoteModeCmd<32 
	 AND Cfg_ModeTransitions[Sts_ModeCurrent].30 AND Cfg_ModeTransitions[Inp_RemoteModeCmd].30 THEN
		Sts_ModeCurrent:=Inp_RemoteModeCmd;
		Cmd_Mode:=Sts_ModeCurrent;
	END_IF
	IF Cmd_Mode<>Sts_ModeCurrent AND Cmd_Mode>1 AND Cmd_Mode<32 
	 AND Cfg_ModeTransitions[Sts_ModeCurrent].30 AND Cfg_ModeTransitions[Cmd_Mode].30 THEN	
		Sts_ModeCurrent:=Cmd_Mode;
	END_IF
END_IF
IF Sts_StateCurrent=31 THEN
	IF RemoteCmdchangerequested AND inp_remoteModeCmd<>0 AND Inp_RemoteModeCmd>1 AND Inp_RemoteModeCmd<32 
	 AND Cfg_ModeTransitions[Sts_ModeCurrent].31 AND Cfg_ModeTransitions[Inp_RemoteModeCmd].31 THEN
		Sts_ModeCurrent:=Inp_RemoteModeCmd;
		Cmd_Mode:=Sts_ModeCurrent;
	END_IF
	IF Cmd_Mode<>Sts_ModeCurrent AND Cmd_Mode>1 AND Cmd_Mode<32 
	 AND Cfg_ModeTransitions[Sts_ModeCurrent].31 AND Cfg_ModeTransitions[Cmd_Mode].31 THEN	
		Sts_ModeCurrent:=Cmd_Mode;
	END_IF
END_IF

ACTION ACT:
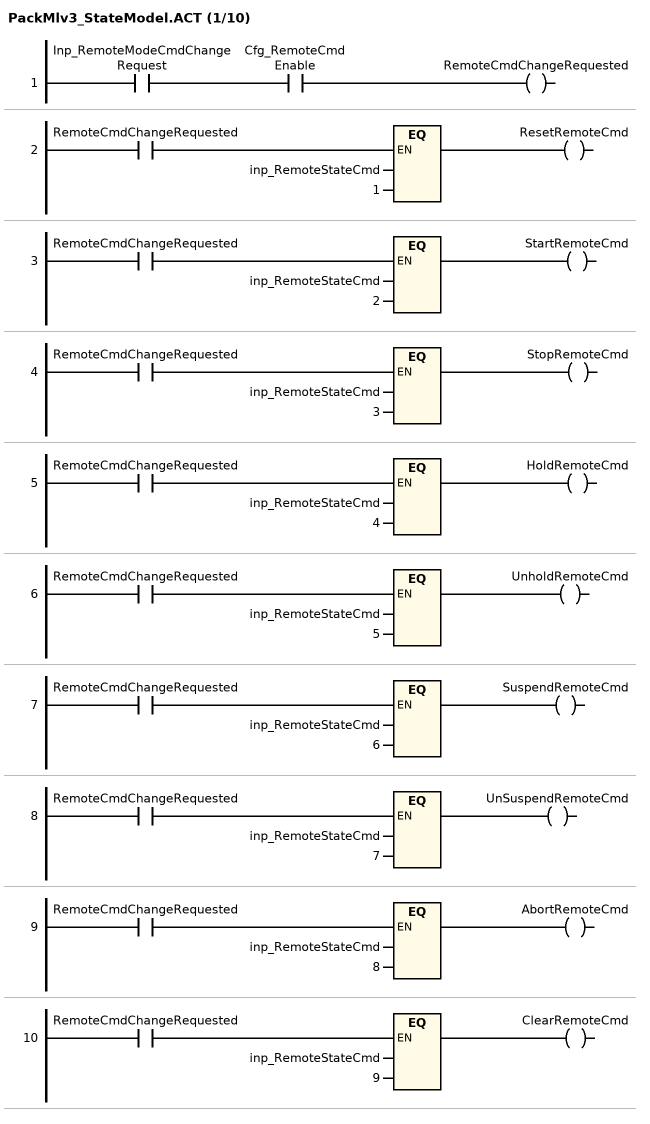
// NETWORK 1
RemoteCmdChangeRequested := Inp_RemoteModeCmdChangeRequest AND Cfg_RemoteCmdEnable;

// NETWORK 2
ResetRemoteCmd := RemoteCmdChangeRequested AND inp_RemoteStateCmd = 1;

// NETWORK 3
StartRemoteCmd := RemoteCmdChangeRequested AND inp_RemoteStateCmd = 2;

// NETWORK 4
StopRemoteCmd := RemoteCmdChangeRequested AND inp_RemoteStateCmd = 3;

// NETWORK 5
HoldRemoteCmd := RemoteCmdChangeRequested AND inp_RemoteStateCmd = 4;

// NETWORK 6
UnholdRemoteCmd := RemoteCmdChangeRequested AND inp_RemoteStateCmd = 5;

// NETWORK 7
SuspendRemoteCmd := RemoteCmdChangeRequested AND inp_RemoteStateCmd = 6;

// NETWORK 8
UnSuspendRemoteCmd := RemoteCmdChangeRequested AND inp_RemoteStateCmd = 7;

// NETWORK 9
AbortRemoteCmd := RemoteCmdChangeRequested AND inp_RemoteStateCmd = 8;

// NETWORK 10
ClearRemoteCmd := RemoteCmdChangeRequested AND inp_RemoteStateCmd = 9;

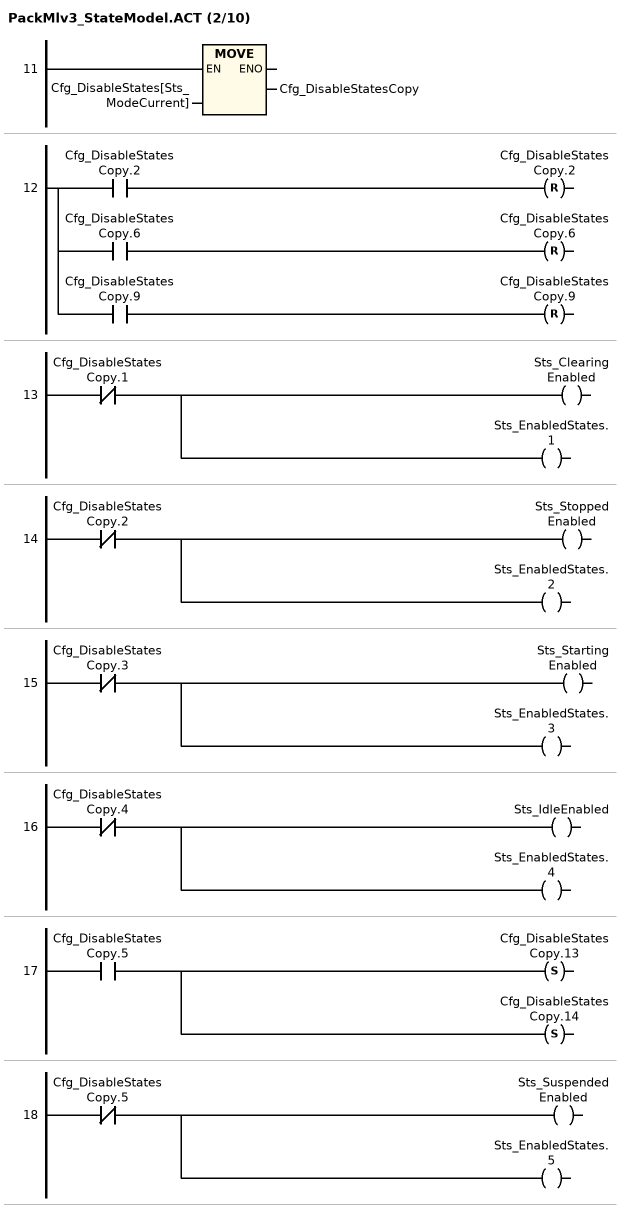
// NETWORK 11
Cfg_DisableStatesCopy := Cfg_DisableStates[Sts_ModeCurrent];

// NETWORK 12
Cfg_DisableStatesCopy.2 R= Cfg_DisableStatesCopy.2;
Cfg_DisableStatesCopy.6 R= Cfg_DisableStatesCopy.6;
Cfg_DisableStatesCopy.9 R= Cfg_DisableStatesCopy.9;

// NETWORK 13
_w1 := NOT Cfg_DisableStatesCopy.1;
Sts_ClearingEnabled := _w1;
Sts_EnabledStates.1 := _w1;

// NETWORK 14
_w2 := NOT Cfg_DisableStatesCopy.2;
Sts_StoppedEnabled := _w2;
Sts_EnabledStates.2 := _w2;

// NETWORK 15
_w3 := NOT Cfg_DisableStatesCopy.3;
Sts_StartingEnabled := _w3;
Sts_EnabledStates.3 := _w3;

// NETWORK 16
_w4 := NOT Cfg_DisableStatesCopy.4;
Sts_IdleEnabled := _w4;
Sts_EnabledStates.4 := _w4;

// NETWORK 17
_w5 := Cfg_DisableStatesCopy.5;
Cfg_DisableStatesCopy.13 S= _w5;
Cfg_DisableStatesCopy.14 S= _w5;

// NETWORK 18
_w6 := NOT Cfg_DisableStatesCopy.5;
Sts_SuspendedEnabled := _w6;
Sts_EnabledStates.5 := _w6;

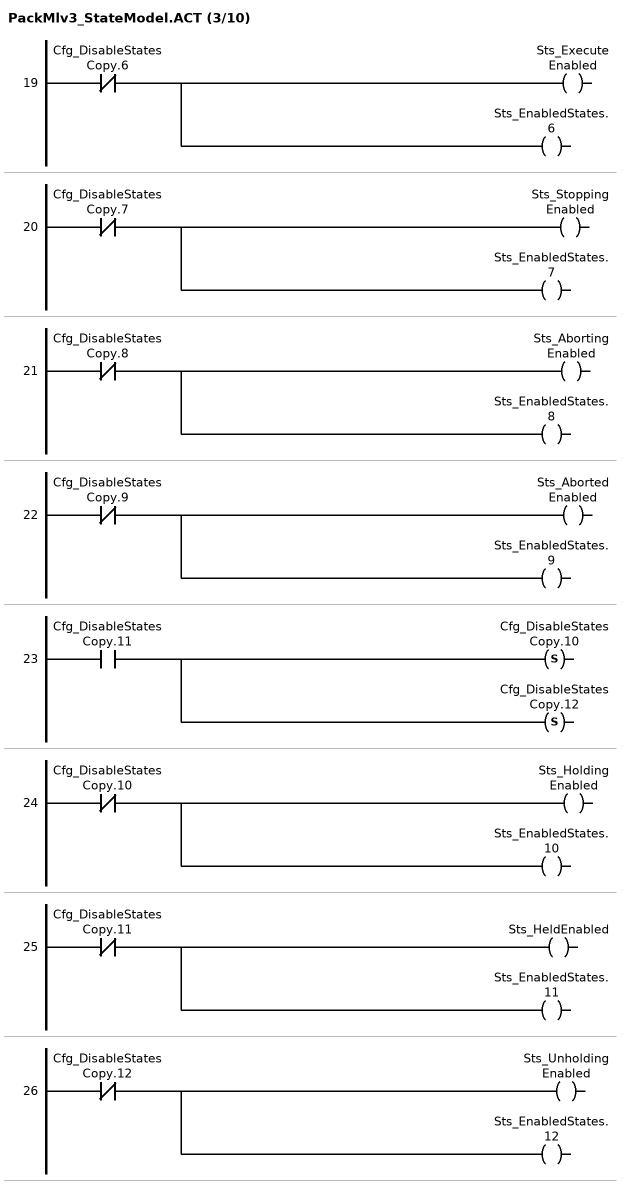
// NETWORK 19
_w7 := NOT Cfg_DisableStatesCopy.6;
Sts_ExecuteEnabled := _w7;
Sts_EnabledStates.6 := _w7;

// NETWORK 20
_w8 := NOT Cfg_DisableStatesCopy.7;
Sts_StoppingEnabled := _w8;
Sts_EnabledStates.7 := _w8;

// NETWORK 21
_w9 := NOT Cfg_DisableStatesCopy.8;
Sts_AbortingEnabled := _w9;
Sts_EnabledStates.8 := _w9;

// NETWORK 22
_w10 := NOT Cfg_DisableStatesCopy.9;
Sts_AbortedEnabled := _w10;
Sts_EnabledStates.9 := _w10;

// NETWORK 23
_w11 := Cfg_DisableStatesCopy.11;
Cfg_DisableStatesCopy.10 S= _w11;
Cfg_DisableStatesCopy.12 S= _w11;

// NETWORK 24
_w12 := NOT Cfg_DisableStatesCopy.10;
Sts_HoldingEnabled := _w12;
Sts_EnabledStates.10 := _w12;

// NETWORK 25
_w13 := NOT Cfg_DisableStatesCopy.11;
Sts_HeldEnabled := _w13;
Sts_EnabledStates.11 := _w13;

// NETWORK 26
_w14 := NOT Cfg_DisableStatesCopy.12;
Sts_UnholdingEnabled := _w14;
Sts_EnabledStates.12 := _w14;

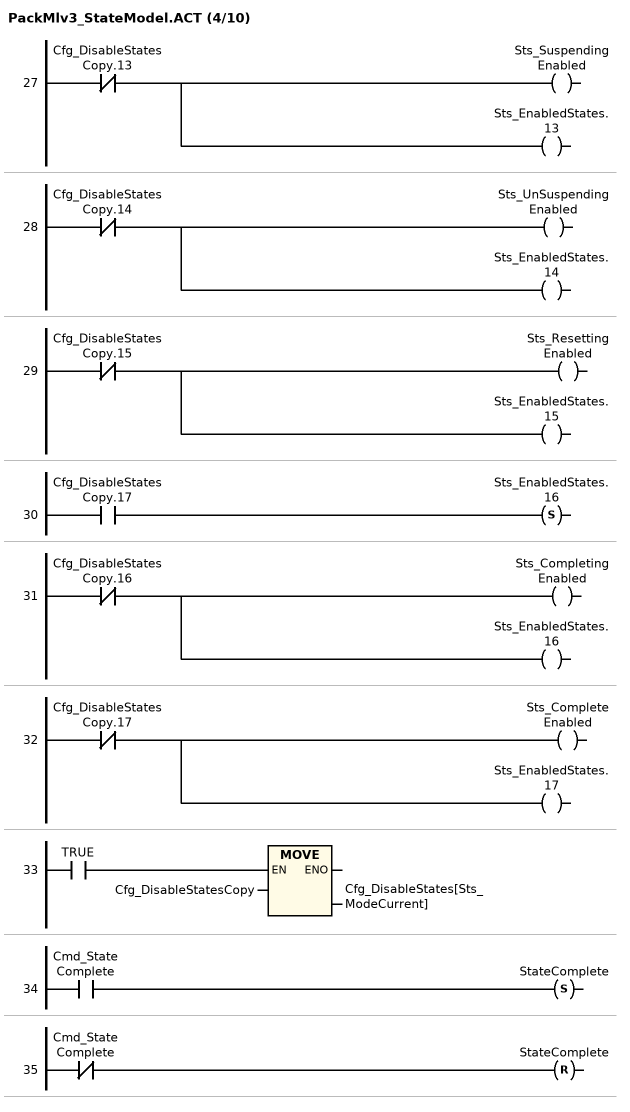
// NETWORK 27
_w15 := NOT Cfg_DisableStatesCopy.13;
Sts_SuspendingEnabled := _w15;
Sts_EnabledStates.13 := _w15;

// NETWORK 28
_w16 := NOT Cfg_DisableStatesCopy.14;
Sts_UnSuspendingEnabled := _w16;
Sts_EnabledStates.14 := _w16;

// NETWORK 29
_w17 := NOT Cfg_DisableStatesCopy.15;
Sts_ResettingEnabled := _w17;
Sts_EnabledStates.15 := _w17;

// NETWORK 30
Sts_EnabledStates.16 S= Cfg_DisableStatesCopy.17;

// NETWORK 31
_w18 := NOT Cfg_DisableStatesCopy.16;
Sts_CompletingEnabled := _w18;
Sts_EnabledStates.16 := _w18;

// NETWORK 32
_w19 := NOT Cfg_DisableStatesCopy.17;
Sts_CompleteEnabled := _w19;
Sts_EnabledStates.17 := _w19;

// NETWORK 33
Cfg_DisableStates[Sts_ModeCurrent] := Cfg_DisableStatesCopy;

// NETWORK 34
StateComplete S= Cmd_StateComplete;

// NETWORK 35
StateComplete R= NOT Cmd_StateComplete;

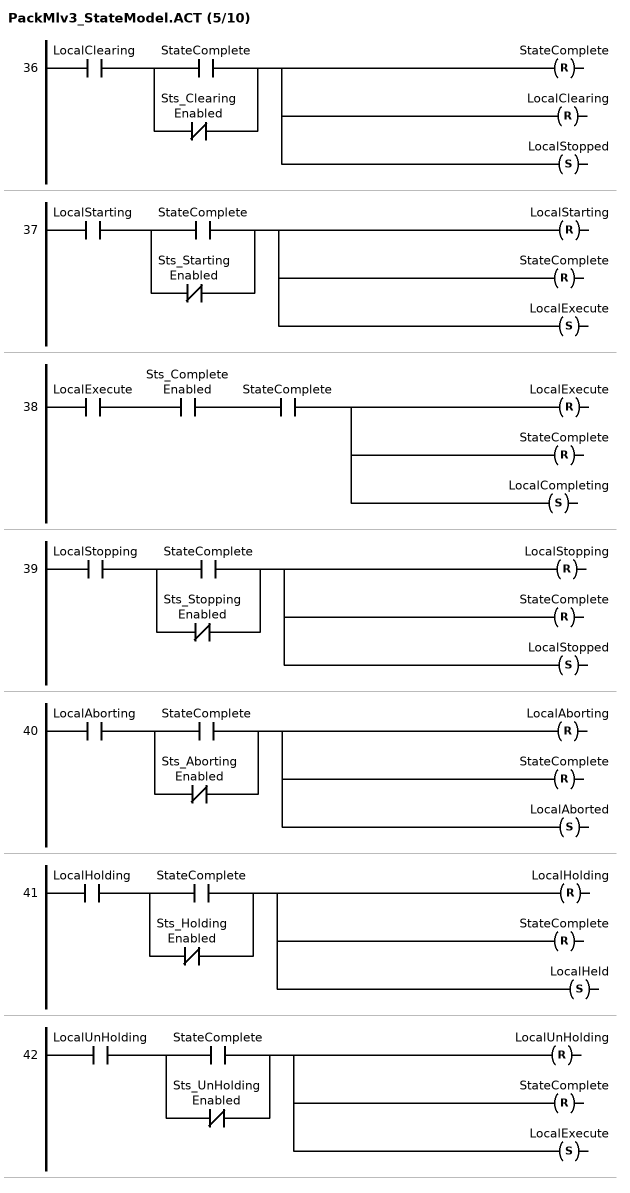
// NETWORK 36
_w20 := LocalClearing AND (StateComplete OR NOT Sts_ClearingEnabled);
StateComplete R= _w20;
LocalClearing R= _w20;
LocalStopped S= _w20;

// NETWORK 37
_w21 := LocalStarting AND (StateComplete OR NOT Sts_StartingEnabled);
LocalStarting R= _w21;
StateComplete R= _w21;
LocalExecute S= _w21;

// NETWORK 38
_w22 := LocalExecute AND Sts_CompleteEnabled AND StateComplete;
LocalExecute R= _w22;
StateComplete R= _w22;
LocalCompleting S= _w22;

// NETWORK 39
_w23 := LocalStopping AND (StateComplete OR NOT Sts_StoppingEnabled);
LocalStopping R= _w23;
StateComplete R= _w23;
LocalStopped S= _w23;

// NETWORK 40
_w24 := LocalAborting AND (StateComplete OR NOT Sts_AbortingEnabled);
LocalAborting R= _w24;
StateComplete R= _w24;
LocalAborted S= _w24;

// NETWORK 41
_w25 := LocalHolding AND (StateComplete OR NOT Sts_HoldingEnabled);
LocalHolding R= _w25;
StateComplete R= _w25;
LocalHeld S= _w25;

// NETWORK 42
_w26 := LocalUnHolding AND (StateComplete OR NOT Sts_UnHoldingEnabled);
LocalUnHolding R= _w26;
StateComplete R= _w26;
LocalExecute S= _w26;

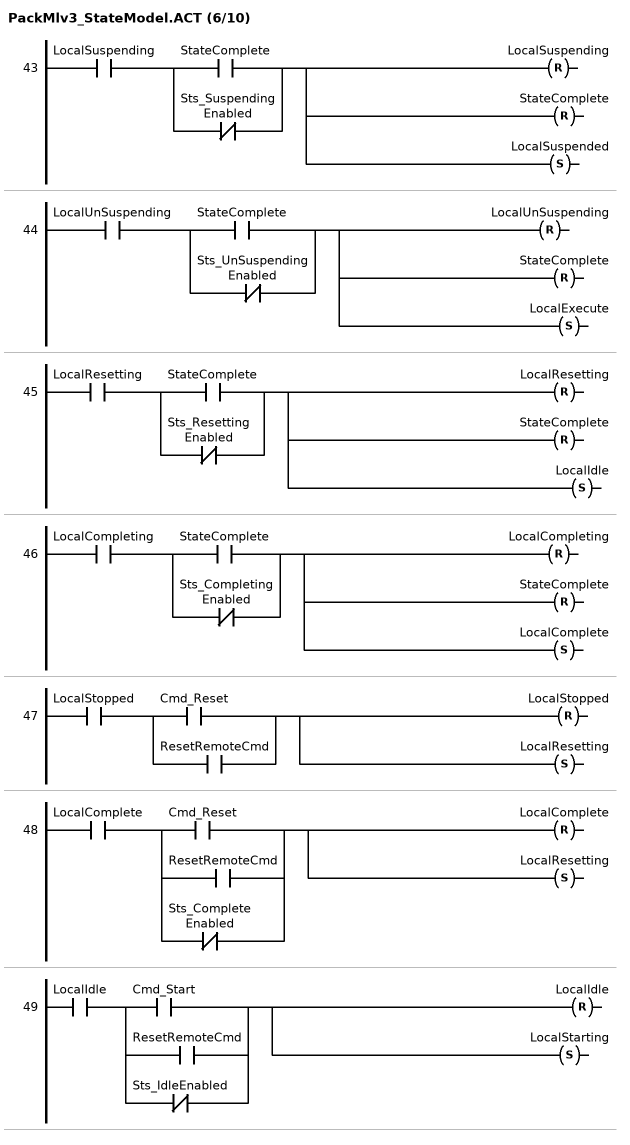
// NETWORK 43
_w27 := LocalSuspending AND (StateComplete OR NOT Sts_SuspendingEnabled);
LocalSuspending R= _w27;
StateComplete R= _w27;
LocalSuspended S= _w27;

// NETWORK 44
_w28 := LocalUnSuspending AND (StateComplete OR NOT Sts_UnSuspendingEnabled);
LocalUnSuspending R= _w28;
StateComplete R= _w28;
LocalExecute S= _w28;

// NETWORK 45
_w29 := LocalResetting AND (StateComplete OR NOT Sts_ResettingEnabled);
LocalResetting R= _w29;
StateComplete R= _w29;
LocalIdle S= _w29;

// NETWORK 46
_w30 := LocalCompleting AND (StateComplete OR NOT Sts_CompletingEnabled);
LocalCompleting R= _w30;
StateComplete R= _w30;
LocalComplete S= _w30;

// NETWORK 47
_w31 := LocalStopped AND (Cmd_Reset OR ResetRemoteCmd);
LocalStopped R= _w31;
LocalResetting S= _w31;

// NETWORK 48
_w32 := LocalComplete AND (Cmd_Reset OR ResetRemoteCmd OR NOT Sts_CompleteEnabled);
LocalComplete R= _w32;
LocalResetting S= _w32;

// NETWORK 49
_w33 := LocalIdle AND (Cmd_Start OR ResetRemoteCmd OR NOT Sts_IdleEnabled);
LocalIdle R= _w33;
LocalStarting S= _w33;

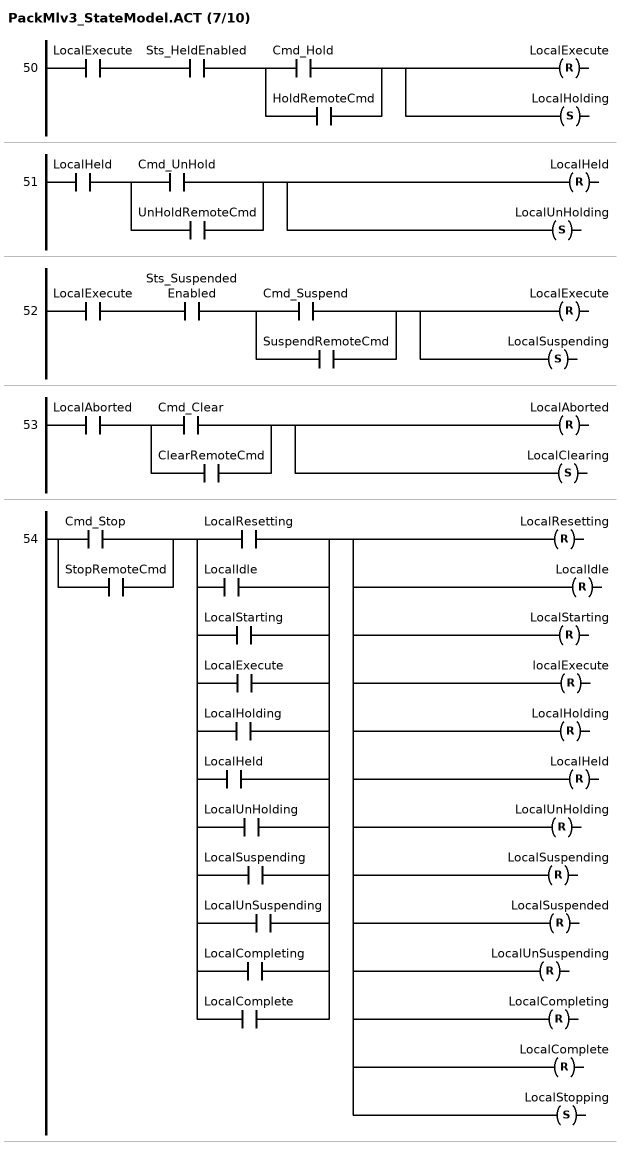
// NETWORK 50
_w34 := LocalExecute AND Sts_HeldEnabled AND (Cmd_Hold OR HoldRemoteCmd);
LocalExecute R= _w34;
LocalHolding S= _w34;

// NETWORK 51
_w35 := LocalHeld AND (Cmd_UnHold OR UnHoldRemoteCmd);
LocalHeld R= _w35;
LocalUnHolding S= _w35;

// NETWORK 52
_w36 := LocalExecute AND Sts_SuspendedEnabled AND (Cmd_Suspend OR SuspendRemoteCmd);
LocalExecute R= _w36;
LocalSuspending S= _w36;

// NETWORK 53
_w37 := LocalAborted AND (Cmd_Clear OR ClearRemoteCmd);
LocalAborted R= _w37;
LocalClearing S= _w37;

// NETWORK 54
_w38 := (Cmd_Stop OR StopRemoteCmd) AND (LocalResetting OR LocalIdle OR LocalStarting OR LocalExecute OR LocalHolding OR LocalHeld OR LocalUnHolding OR LocalSuspending OR LocalUnSuspending OR LocalCompleting OR LocalComplete);
LocalResetting R= _w38;
LocalIdle R= _w38;
LocalStarting R= _w38;
localExecute R= _w38;
LocalHolding R= _w38;
LocalHeld R= _w38;
LocalUnHolding R= _w38;
LocalSuspending R= _w38;
LocalSuspended R= _w38;
LocalUnSuspending R= _w38;
LocalCompleting R= _w38;
LocalComplete R= _w38;
LocalStopping S= _w38;

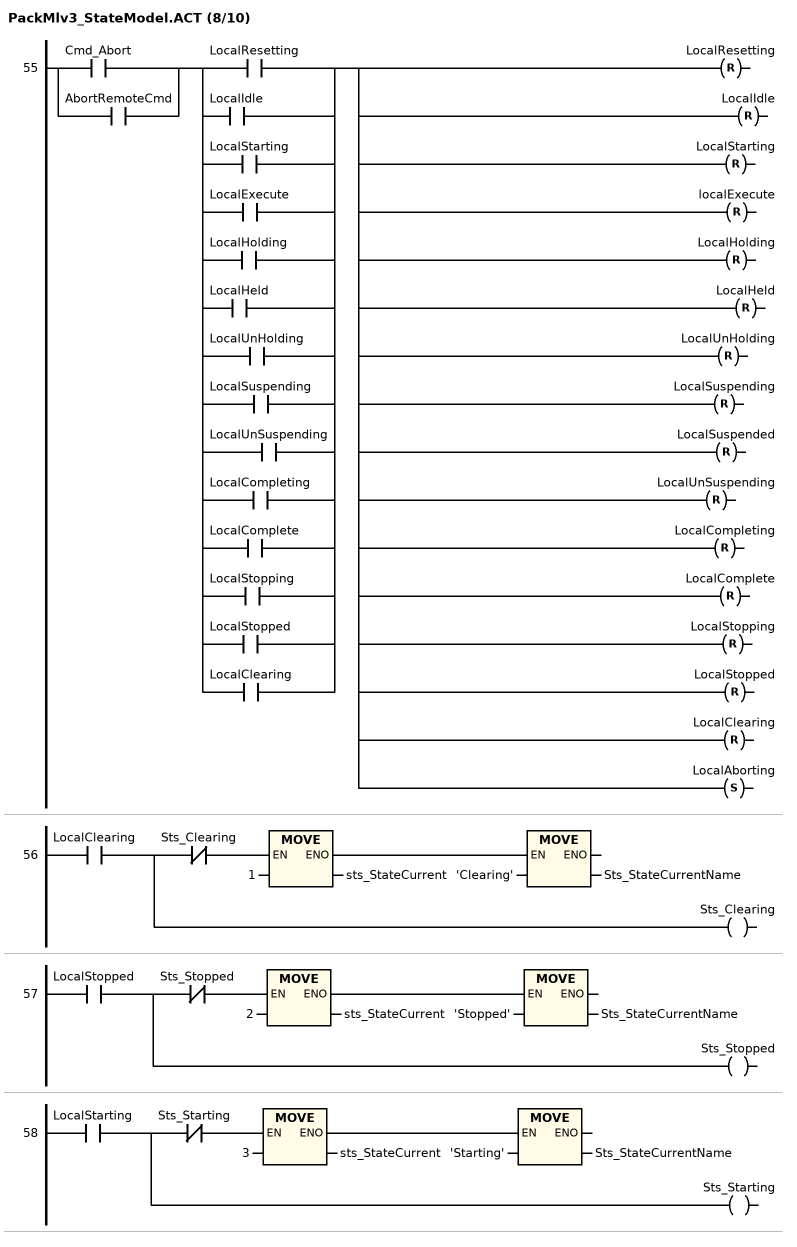
// NETWORK 55
_w39 := (Cmd_Abort OR AbortRemoteCmd) AND (LocalResetting OR LocalIdle OR LocalStarting OR LocalExecute OR LocalHolding OR LocalHeld OR LocalUnHolding OR LocalSuspending OR LocalUnSuspending OR LocalCompleting OR LocalComplete OR LocalStopping OR LocalStopped OR LocalClearing);
LocalResetting R= _w39;
LocalIdle R= _w39;
LocalStarting R= _w39;
localExecute R= _w39;
LocalHolding R= _w39;
LocalHeld R= _w39;
LocalUnHolding R= _w39;
LocalSuspending R= _w39;
LocalSuspended R= _w39;
LocalUnSuspending R= _w39;
LocalCompleting R= _w39;
LocalComplete R= _w39;
LocalStopping R= _w39;
LocalStopped R= _w39;
LocalClearing R= _w39;
LocalAborting S= _w39;

// NETWORK 56
_w40 := LocalClearing AND NOT Sts_Clearing;
IF _w40 THEN sts_StateCurrent := 1; END_IF
IF _w40 THEN Sts_StateCurrentName := 'Clearing'; END_IF
Sts_Clearing := LocalClearing;

// NETWORK 57
_w41 := LocalStopped AND NOT Sts_Stopped;
IF _w41 THEN sts_StateCurrent := 2; END_IF
IF _w41 THEN Sts_StateCurrentName := 'Stopped'; END_IF
Sts_Stopped := LocalStopped;

// NETWORK 58
_w42 := LocalStarting AND NOT Sts_Starting;
IF _w42 THEN sts_StateCurrent := 3; END_IF
IF _w42 THEN Sts_StateCurrentName := 'Starting'; END_IF
Sts_Starting := LocalStarting;

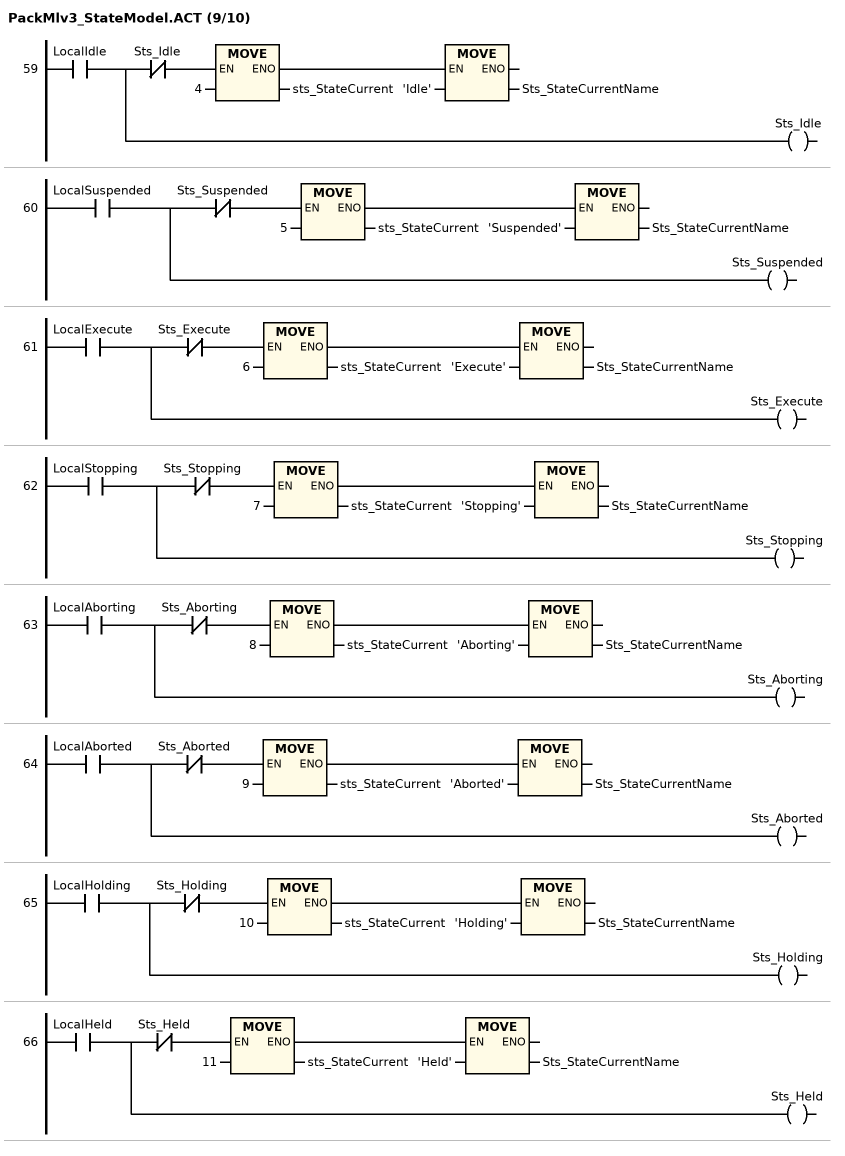
// NETWORK 59
_w43 := LocalIdle AND NOT Sts_Idle;
IF _w43 THEN sts_StateCurrent := 4; END_IF
IF _w43 THEN Sts_StateCurrentName := 'Idle'; END_IF
Sts_Idle := LocalIdle;

// NETWORK 60
_w44 := LocalSuspended AND NOT Sts_Suspended;
IF _w44 THEN sts_StateCurrent := 5; END_IF
IF _w44 THEN Sts_StateCurrentName := 'Suspended'; END_IF
Sts_Suspended := LocalSuspended;

// NETWORK 61
_w45 := LocalExecute AND NOT Sts_Execute;
IF _w45 THEN sts_StateCurrent := 6; END_IF
IF _w45 THEN Sts_StateCurrentName := 'Execute'; END_IF
Sts_Execute := LocalExecute;

// NETWORK 62
_w46 := LocalStopping AND NOT Sts_Stopping;
IF _w46 THEN sts_StateCurrent := 7; END_IF
IF _w46 THEN Sts_StateCurrentName := 'Stopping'; END_IF
Sts_Stopping := LocalStopping;

// NETWORK 63
_w47 := LocalAborting AND NOT Sts_Aborting;
IF _w47 THEN sts_StateCurrent := 8; END_IF
IF _w47 THEN Sts_StateCurrentName := 'Aborting'; END_IF
Sts_Aborting := LocalAborting;

// NETWORK 64
_w48 := LocalAborted AND NOT Sts_Aborted;
IF _w48 THEN sts_StateCurrent := 9; END_IF
IF _w48 THEN Sts_StateCurrentName := 'Aborted'; END_IF
Sts_Aborted := LocalAborted;

// NETWORK 65
_w49 := LocalHolding AND NOT Sts_Holding;
IF _w49 THEN sts_StateCurrent := 10; END_IF
IF _w49 THEN Sts_StateCurrentName := 'Holding'; END_IF
Sts_Holding := LocalHolding;

// NETWORK 66
_w50 := LocalHeld AND NOT Sts_Held;
IF _w50 THEN sts_StateCurrent := 11; END_IF
IF _w50 THEN Sts_StateCurrentName := 'Held'; END_IF
Sts_Held := LocalHeld;

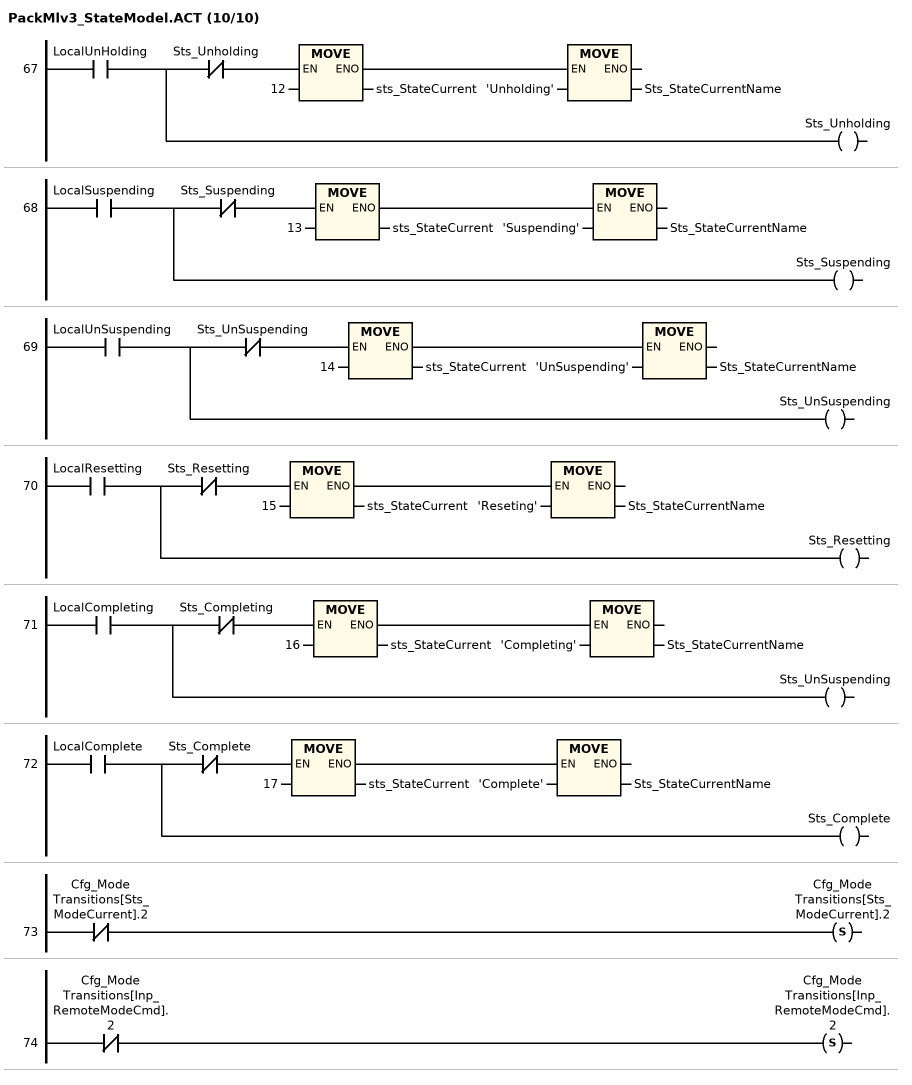
// NETWORK 67
_w51 := LocalUnHolding AND NOT Sts_Unholding;
IF _w51 THEN sts_StateCurrent := 12; END_IF
IF _w51 THEN Sts_StateCurrentName := 'Unholding'; END_IF
Sts_Unholding := LocalUnHolding;

// NETWORK 68
_w52 := LocalSuspending AND NOT Sts_Suspending;
IF _w52 THEN sts_StateCurrent := 13; END_IF
IF _w52 THEN Sts_StateCurrentName := 'Suspending'; END_IF
Sts_Suspending := LocalSuspending;

// NETWORK 69
_w53 := LocalUnSuspending AND NOT Sts_UnSuspending;
IF _w53 THEN sts_StateCurrent := 14; END_IF
IF _w53 THEN Sts_StateCurrentName := 'UnSuspending'; END_IF
Sts_UnSuspending := LocalUnSuspending;

// NETWORK 70
_w54 := LocalResetting AND NOT Sts_Resetting;
IF _w54 THEN sts_StateCurrent := 15; END_IF
IF _w54 THEN Sts_StateCurrentName := 'Reseting'; END_IF
Sts_Resetting := LocalResetting;

// NETWORK 71
_w55 := LocalCompleting AND NOT Sts_Completing;
IF _w55 THEN sts_StateCurrent := 16; END_IF
IF _w55 THEN Sts_StateCurrentName := 'Completing'; END_IF
Sts_UnSuspending := LocalCompleting;

// NETWORK 72
_w56 := LocalComplete AND NOT Sts_Complete;
IF _w56 THEN sts_StateCurrent := 17; END_IF
IF _w56 THEN Sts_StateCurrentName := 'Complete'; END_IF
Sts_Complete := LocalComplete;

// NETWORK 73
Cfg_ModeTransitions[Sts_ModeCurrent].2 S= NOT Cfg_ModeTransitions[Sts_ModeCurrent].2;

// NETWORK 74
Cfg_ModeTransitions[Inp_RemoteModeCmd].2 S= NOT Cfg_ModeTransitions[Inp_RemoteModeCmd].2;
END_ACTION

END_FUNCTION_BLOCK

// ---- Add-On-Instructions/AOI_CylinderAdmin.TcPOU
FUNCTION_BLOCK AOI_CylinderAdmin
VAR_INPUT
END_VAR
VAR_OUTPUT
	ActInTime: DINT;
	ActOutTime: DINT;
END_VAR
VAR
	TON_InCheck: TON;
	TON_OutCheck: TON;
	rtOUT: R_trig;
    rtIn: R_trig;
END_VAR
VAR_IN_OUT
	Admin: UDT_CylinderAdmin;
END_VAR

IF admin.i.mode=0 THEN
   IF admin.i.HmiIN THEN
	  admin.o.ValveIn:=TRUE;
	  admin.o.ValveOut:=FALSE;
   END_IF
   IF admin.i.HmiOUT THEN
	  admin.o.ValveIn:=FALSE;
	  admin.o.ValveOut:=TRUE;
   END_IF
END_IF
IF admin.i.mode=1 THEN
   IF admin.i.ActiveIn THEN
	  admin.o.ValveIn:=TRUE;
	  admin.o.ValveOut:=FALSE;
   END_IF
   IF admin.i.ActiveOut THEN
	  admin.o.ValveIn:=FALSE;
	  admin.o.ValveOut:=TRUE;
   END_IF
   IF NOT admin.i.ActiveIn AND NOT admin.i.ActiveOut  THEN
	  admin.o.ValveIn:=FALSE;
	  admin.o.ValveOut:=FALSE;
   END_IF
END_IF

TON_InCheck(IN:=admin.o.ValveIn AND NOT admin.i.Reset , PT:=DINT_TO_TIME(admin.i.CheckTime) , Q=> , ET=> );
TON_OutCheck(IN:=admin.o.ValveOut AND NOT admin.i.Reset, PT:=DINT_TO_TIME(admin.i.CheckTime) , Q=> , ET=> );
IF ton_incheck.Q AND NOT admin.i.InSensor THEN
   admin.o.Error:=TRUE;
END_IF
IF Ton_OutCheck.Q AND NOT admin.i.OutSensor THEN 
   admin.o.Error:=TRUE;
END_IF
IF admin.i.Reset THEN
   admin.o.Error:=FALSE;
END_IF

IF rtOUT.Q  AND NOT admin.o.Error THEN
   ActOutTime:=TIME_TO_DINT(TON_OutCheck.ET);
END_IF

IF rtIN.Q  AND NOT admin.o.Error THEN
   ActInTime:=TIME_TO_DINT(TON_InCheck.ET);
END_IF

rtOUT(CLK:= admin.i.OutSensor , Q=> );
rtIn(CLK:=  admin.i.InSensor, Q=> );

END_FUNCTION_BLOCK

// ---- Add-On-Instructions/AOI_VacuumAdmin.TcPOU
FUNCTION_BLOCK AOI_VacuumAdmin
VAR_INPUT
END_VAR
VAR_OUTPUT
END_VAR
VAR_IN_OUT
	admin: UDT_VacuumAdmin;
END_VAR

VAR
	ftVacuum: F_trig;
	tonBlow: TON;
	tonCheck: TON;	
END_VAR

IF admin.i.ActiveIN THEN
	admin.o.ValveIn:=TRUE;
	ELSE 
	admin.o.ValveIn:=FALSE;
END_IF

ftVacuum(CLK:=admin.o.ValveIn , Q=> );
IF ftVacuum.Q THEN
   admin.o.ValveOut:=TRUE;
END_IF
IF tonBlow.Q THEN
   admin.o.ValveOut:=FALSE;
END_IF

tonBlow(IN:=admin.o.ValveOut, PT:=DINT_TO_TIME(admin.i.BlowTime) , Q=> , ET=> );
tonCheck(IN:=admin.o.ValveIn AND NOT admin.i.reset , PT:=DINT_TO_TIME(admin.i.CheckTime)  , Q=> , ET=> );

IF tonCheck.Q AND NOT admin.i.Sensor THEN
	admin.o.Error :=TRUE;
END_IF

IF admin.i.reset THEN
   admin.o.Error :=FALSE;
END_IF

END_FUNCTION_BLOCK

// ---- Add-On-Instructions/AOI_SensorAdmin.TcPOU
FUNCTION_BLOCK AOI_SensorAdmin
VAR_INPUT
END_VAR
VAR_OUTPUT
END_VAR
VAR
	TON_Fliter: TON;

END_VAR
VAR_IN_OUT
	Admin: UDT_SensorAdmin;
END_VAR

TON_Fliter(IN:= admin.i.Link, PT:=DINT_TO_TIME(admin.i.FilterTime) , Q=>admin.o.Value , ET=> );

END_FUNCTION_BLOCK

// ---- Add-On-Instructions/AOI_HeatBase.TcPOU
FUNCTION_BLOCK AOI_HeatBase
VAR_INPUT
	Enable: BOOL;
	Reset: BOOL;
	PV: REAL;
	SV: REAL;
	HighLimit: REAL;
	LowLimit: REAL;
	MaxLimit: REAL;
	Kp: REAL:=0.8;
	Ki: REAL:=1;
	Kd: REAL:=5;
END_VAR
VAR_OUTPUT
	Active: BOOL;
	Error: BOOL;
	ErrorID: INT;	
END_VAR
VAR
    blinkAct: blink;
	tonLow: Ton;
	tonHigh: Ton;	
	iDiff: INT;
	arDiff: ARRAY[0..255] OF REAL;
	i: INT;
	n: INT;
	tonSample: Ton;
	rAverageDiff: REAL;
	rSumDiff: REAL;
	j: INT;
	iAct: INT;
	iPID: INT;
	arM: ARRAY[0..255] OF REAL;

	arPV: ARRAY[0..255] OF REAL;
	Mi: REAL;
	MX:REAL;
	Kc: INT:=8;
END_VAR

(*
IF PV < SV AND NOT ErrorID.0 AND NOT ErrorID.1 THEN
	Active:=TRUE;
ELSE 
	Active:=FALSE;
END_IF	  
*)

tonHigh(IN:=(PV> SV+HighLimit) , PT:= T#3S, Q=> , ET=> );
IF tonHigh.Q THEN
	Error:=TRUE;
	ErrorID.0:=TRUE;
END_IF

IF PV>MaxLimit THEN
	Error:=TRUE;        
	ErrorID.1:=TRUE;		
END_IF       

tonLow(IN:=(PV < SV-Lowlimit) , PT:= T#3S, Q=> , ET=> );
IF tonLow.Q THEN
	Error:=TRUE;     
	ErrorID.2:=TRUE;	  
END_IF

IF Reset THEN
	Error:=FALSE;
	ErrorID:=0;
END_IF

CASE iDiff OF
	0:
	  IF Enable THEN
		  iDiff:=1;
	  END_IF
	1:  
	  IF SV>0 THEN
		  IF PV < SV-SV*0.05 THEN
			 iDiff:=100; 
		  END_IF
		  IF PV > SV-SV*0.05 AND NOT ErrorID.0 AND NOT ErrorID.1 THEN
			 rSumDiff:=0;		  
			 iDiff:=10;
		  END_IF
	  END_IF 
	10:
	  arDiff[i]:=SV-PV;
	  IF ABS(arDiff[i]>SV) THEN
		  arDiff[i]:=0;
	  END_IF
	  rSumDiff:=rSumDiff+arDiff[i];
	  (*
	  IF i = Kc THEN
	     rSumDiff:= 0;
	     FOR j:=0 TO Kc DO
		     rSumDiff:= rSumDiff+ arDiff[j];
			 rAverageDiff:=rSumDiff/Kc;
	     END_FOR
	  END_IF  
	  *)
	  iDiff:=20;
	 
    20: 
      arM[0]:=Kp*arDiff[i];
      arM[1]:= Ki*rSumDiff;
	  IF arM[1]>1900 THEN
		 arM[1]:=1900;
	  END_IF
	  IF arM[1]<-1900 THEN
		 arM[1]:=-1900;
	  END_IF
	  
	  IF i=0 THEN
         arM[2]:=Kd*(arDiff[i]-arDiff[Kc]);
	  ELSE
	     arM[2]:=Kd*(arDiff[i]-arDiff[i-1]);
	  END_IF 
	  arM[2]:=arM[2];

	  arM[3]:= (arM[0]+arM[1]+arM[2])*100;
	  IF ARM[3]>1800 THEN
		 ARM[3]:=1800;
		 ELSE IF ARM[3]<200 THEN
			     ARM[3]:=200;
		      END_IF
	  END_IF	
	  iDiff:=30;
	  
	30:  
	  Active:=TRUE;
	  tonSample(IN:= TRUE, PT:= REAL_TO_TIME(arM[3]), Q=> , ET=> );
	  IF tonSample.Q THEN
		  tonSample(IN:= FALSE, PT:= REAL_TO_TIME(arM[3]), Q=> , ET=> );
		  Active:=FALSE;
		  iDiff:=40;
	  END_IF
	40:
	  Active:=FALSE;
	  tonSample(IN:= TRUE, PT:= REAL_TO_TIME(2000-arM[3]), Q=> , ET=> );
	  IF tonSample.Q THEN
		  tonSample(IN:= FALSE, PT:= REAL_TO_TIME(2000-arM[3]), Q=> , ET=> );
		  Active:=FALSE;
		  iDiff:=50;
	  END_IF

	50:  
	  i:=i+1;
	  IF i>Kc THEN
		  i:=0;  
	  END_IF	   
	  iDiff:=0;
	  
	100: 
		IF PV < SV-SV*0.05 AND NOT ErrorID.0 AND NOT ErrorID.1 THEN
			Active:=TRUE;
		ELSE 
			Active:=FALSE;
			iDiff:=0;
		END_IF	  
	  	 
END_CASE

CASE iAct OF 
	0:iAct:=0;
	
END_CASE

END_FUNCTION_BLOCK

// ---- Add-On-Instructions/AOI_Timer.TcPOU
FUNCTION_BLOCK AOI_Timer
VAR_INPUT
	bEnable: BOOL;
	bReset: BOOL;
END_VAR
VAR_OUTPUT
	diSecond:DINT;
	diMinute: DINT;
	diHour: DINT;
	diTotalSecond: DINT;
	diTotalMinute: DINT;
	diTotalHour: DINT;
END_VAR
VAR
	tonSecond: Ton;
END_VAR

tonSecond(IN:= bEnable AND NOT tonSecond.Q, PT:=T#1000MS , Q=> , ET=> );
IF tonSecond.Q THEN
	diSecond:=diSecond+1;
	diTotalSecond:=diTotalSecond+1;
END_IF

IF diSecond>59 THEN
	diSecond:=0;
	diMinute:=diMinute+1;
	diTotalMinute:=diTotalMinute+1;
END_IF

IF diMinute>59 THEN
	diMinute:=0;
	diHour:=diHour+1;
	diTotalHour:=diTotalHour+1;
END_IF

IF bReset THEN
	diSecond :=0;
	diMinute:=0;
	diHour:=0;
	diTotalSecond:=0;
	diTotalMinute:=0;
	diTotalHour:=0;	
END_IF

END_FUNCTION_BLOCK

// ---- POUs/PackMaL_UN01/EM01_Master.TcPOU
PROGRAM EM01_Master
VAR
	ref_Master1: REFERENCE TO UDT_AXISADMIN;	
	ref_Follower4: REFERENCE TO UDT_AXISADMIN;
	ref_Follower5: REFERENCE TO UDT_AXISADMIN;	
	Ref_MachineStateModel: REFERENCE TO PackMlv3_StateModel;
	ref_Work_Recipe: REFERENCE TO UDT_Hmi_Output; //当前生产的配方

    Ref_Unit: REFERENCE TO UDT_UnitAdmin;
	ref_lrLatchMasterPos: REFERENCE TO LREAL;
	ref_BinList: REFERENCE TO UDT_BINlist;	
	ref_diBeltObjCnt: REFERENCE TO DINT;
	EM_No: INT:=1;

	tonAbortingWatchDog: TON;   
	MasterSeq: SequenceTransfer;
	
END_VAR

VAR CONSTANT

END_VAR

// 主轴走200MM产出一个产品
Ref_MachineStateModel REF= UN01_MachineStateModel;
Ref_Unit REF=Unit01;
ref_Work_Recipe REF= HMI_Output;
ref_Follower4  REF= arRealAxisAdmin[44];
ref_Follower5  REF= arRealAxisAdmin[45];
ref_Master1 REF= arVirtualAxisAdmin[1];

ref_BinList REF=Glb_BinList;
ref_diBeltObjCnt REF=glb_diBeltObjCnt;
CM01_Master();
MainRoution();
SR99_FaultHandle();

ref_master1.i.PosRangeTable[1][1]:=190;
ref_master1.i.PosRangeTable[1][2]:=200;

ACTION CM01_Master:
CASE MasterSeq.Now OF		 
	0: 
	   IF Ref_MachineStateModel.Sts_Resetting THEN
		  MasterSeq(ExeCute:= TRUE, Next:= Seq_Resetting );
	   END_IF	   
	   IF Ref_MachineStateModel.Sts_Stopping  THEN
          MasterSeq(ExeCute:= TRUE, Next:= Seq_StoppingDone );  
	   END_IF	

	Seq_Resetting:
		IF NOT ref_Master1.o.PowerOn  THEN;
		   ref_Master1.i.Enable:=TRUE;
	    ELSE
		   MasterSeq(ExeCute:= TRUE, Next:= 20 );
		END_IF
	    IF Ref_MachineStateModel.Sts_Stopping  THEN
		   MasterSeq(ExeCute:= TRUE, Next:= Seq_Stopping);  
	    END_IF	
	20:	
	       ref_master1.i.PosRangeTable[1][1]:=0;
		   ref_master1.i.PosRangeTable[1][2]:=10;
		   ref_master1.i.JogAcc:=100;
		   ref_Master1.i.JogDec:=5000;
		   IF NOT glb_AllAxisHomed_UN01 THEN
			  MasterSeq(ExeCute:= TRUE, Next:= 21 );
			  ELSE
			  MasterSeq(ExeCute:= TRUE, Next:= Seq_ResettingDone );
		   END_IF
	21:    
		   ref_Master1.i.HomeMode:=2;
		   ref_Master1.i.Home:=TRUE;
		   IF ref_Master1.o.HomeDone THEN
			   ref_Master1.i.Home:=FALSE;
			   MasterSeq(ExeCute:= TRUE, Next:= 30 );
		   ELSE IF Ref_MachineStateModel.Sts_Stopping  THEN
		           MasterSeq(ExeCute:= TRUE, Next:= Seq_Stopping);  
	            END_IF	 
		   END_IF
    30:   

		  glb_diBeltObjCnt:=0;
          MasterSeq(ExeCute:= TRUE, Next:= Seq_ResettingDone ); 
		  
	Seq_ResettingDone: 
         IF NOT Ref_MachineStateModel.Sts_Resetting THEN
			MasterSeq(ExeCute:= TRUE, Next:= 0 );
		 END_IF	  
 	  
	Seq_Stopping:	
	     MasterSeq(ExeCute:= TRUE, Next:= Seq_StoppingDone); 
	Seq_StoppingDone: 
	     IF NOT Ref_MachineStateModel.Sts_Stopping THEN
			MasterSeq(ExeCute:= TRUE, Next:= 0 );
		 END_IF	   
		 
END_CASE
MasterSeq(ExeCute:= FALSE, Next:= , Last=> , Now=> );
END_ACTION

ACTION MainRoution:
EM_No:=1;
IF Ref_Unit.EM_Selected[EM_No] THEN
	IF Ref_MachineStateModel.Sts_Holding THEN
		Ref_Unit.EM_Holding_Done[EM_No]:=TRUE;
		ELSE
		Ref_Unit.EM_Holding_Done[EM_No]:=FALSE;
	END_IF
	IF Ref_MachineStateModel.Sts_UnHolding THEN
		Ref_Unit.EM_UnHolding_Done[EM_No]:=TRUE;
		ELSE
		Ref_Unit.EM_UnHolding_Done[EM_No]:=FALSE;
	END_IF
	
	IF Ref_MachineStateModel.Sts_Suspending THEN
		Ref_Unit.EM_Suspending_Done[EM_No]:=TRUE;
		ELSE
		Ref_Unit.EM_Suspending_Done[EM_No]:=FALSE;
	END_IF
	
	IF Ref_MachineStateModel.Sts_UnSuspending THEN
		Ref_Unit.EM_UnSuspending_Done[EM_No]:=TRUE;
		ELSE
		Ref_Unit.EM_UnSuspending_Done[EM_No]:=FALSE;
	END_IF
		
	IF Ref_MachineStateModel.Sts_Resetting AND MasterSeq.Now=Seq_ResettingDone  THEN
	   Ref_Unit.EM_Resetting_Done[EM_No]:=TRUE; 
       ELSE   
	   Ref_Unit.EM_Resetting_Done[EM_No]:=FALSE;
	END_IF
	
	IF Ref_MachineStateModel.Sts_Clearing THEN
	      Ref_Unit.EM_Clearing_Done[EM_No]:=TRUE;
		  ELSE
		  Ref_Unit.EM_Clearing_Done[EM_No]:=FALSE;
	END_IF
	
	IF Ref_MachineStateModel.Sts_Aborting THEN
	   MasterSeq(ExeCute:= TRUE, Next:= 0 );
       IF tonAbortingWatchDog.Q THEN
		  ref_Master1.i.Disable:=TRUE;
		  Ref_Unit.EM_Aborting_Done[EM_No]:=TRUE;
	   END_IF
	   ELSE
		  Ref_Unit.EM_Aborting_Done[EM_No]:=FALSE;
	END_IF
	tonAbortingWatchDog(IN:= Ref_MachineStateModel.Sts_Aborting, PT:=T#3S , Q=> , ET=> );
	
	IF Ref_MachineStateModel.Sts_Starting THEN
	   Ref_Unit.EM_Starting_Done[EM_No]:=TRUE;
	   ELSE
	   Ref_Unit.EM_Starting_Done[EM_No]:=FALSE;
	END_IF
	
	IF Ref_MachineStateModel.Sts_Stopping  AND MasterSeq.Now=Seq_StoppingDone THEN
	   Ref_Unit.EM_Stopping_Done[EM_No]:=TRUE;
	   ELSE	   
	   Ref_Unit.EM_Stopping_Done[EM_No]:=FALSE;
	END_IF

END_IF
END_ACTION

ACTION SR99_FaultHandle:
;
END_ACTION

END_PROGRAM

// ---- Add-On-Instructions/SequenceTransfer.TcPOU
FUNCTION_BLOCK SequenceTransfer
VAR_INPUT	
    Execute:BOOL;
	Next: INT;
	Hold: BOOL;
END_VAR
VAR_OUTPUT
	Last: INT;
	Now: INT;
END_VAR
VAR_IN_OUT
END_VAR

IF Execute AND NOT Hold THEN
   Last:=Now;
   Now:=Next;
   Execute:=FALSE;
END_IF

END_FUNCTION_BLOCK

// ---- POUs/PackMaL_UN01/EM02_Follower1.TcPOU
PROGRAM EM02_Follower1
VAR
	ref_Master: REFERENCE TO UDT_AXISADMIN;
	ref_Follower: REFERENCE TO UDT_AXISADMIN;
	Ref_MachineStateModel: REFERENCE TO PackMlv3_StateModel;
	Ref_Unit: REFERENCE TO UDT_UnitAdmin;
	EM_No: INT:=2;
	tonAbortingWatchDog: TON;
	tonStoppingWatchDog: Ton;
	MC_CamIn_Follower: MC_CamIn;

	MC_CamTableSelect_Follower: MC_CamTableSelect;
	CamTableFollower: MC_CAM_REF;
	table1: ARRAY[1..2] OF MC_MotionFunctionPoint; (*用于定义电子凸轮表中的关键点*)

    MC_ReadCamTableSlaveDynamicsFollwer: MC_ReadCamTableSlaveDynamics;

	tonFollowerSeq: TON;
	FollowerSeq: SequenceTransfer;	

	i: INT;
	lrPosCnt: INT;
	bRecipeComplete: BOOL;
	bBeltInRange: BOOL;
	iLastSeq: INT;
	j: INT;
	tonBufferCyclinderDelay: TON;
END_VAR

VAR CONSTANT
	iCamID: MC_CAM_ID:=1;		
END_VAR

//减速比10/1 同步轮周长400 ，皮带总长5200，26个工位，工位间距200

Ref_MachineStateModel REF= UN01_MachineStateModel;
Ref_Unit REF=Unit01;
ref_Master REF= arVirtualAxisAdmin[1];
ref_Follower REF= arRealAxisAdmin[41];
MainRoution();
CM01_Cam();
SR999_Faulthandler();

ACTION CM01_Cam:
//凸轮1曲线
camTableFollower.ArraySize:=SIZEOF(table1);
camTableFollower.NoOfColumns:=1;
camTableFollower.NoOfRows:=2;
camTableFollower.pArray:=ADR(table1);
camTableFollower.TableType:=MC_TABLETYPE_MOTIONFUNCTION;

table1[1].FunctionType:=MOTIONFUNCTYPE_POLYNOM1;
table1[1].MasterPos:=0;
table1[1].SlavePos:=0;
table1[1].PointIndex:=1;
table1[1].PointType:=MOTIONPOINTTYPE_MOTION;
		
table1[2].FunctionType:=MOTIONFUNCTYPE_POLYNOM1;
table1[2].MasterPos:=200;
table1[2].SlavePos:=200;
table1[2].PointIndex:=2;
table1[2].PointType:=MOTIONPOINTTYPE_MOTION;
// 凸轮耦合
MC_CamIn_Follower(
	Master:= ref_Master.Axis, 
	Slave:= ref_Follower.Axis, 
	Execute:= ref_Follower.i.CamIn, 
	MasterOffset:= , 
	SlaveOffset:= , 
	MasterScaling:= 1, 
	SlaveScaling:= 1, 
	StartMode:= MC_STARTMODE_ABSOLUTE, 
	CamTableID:= iCamID, 
	BufferMode:= , 
	Options:= , 
	InSync=> , 
	Busy=> , 
	Active=> , 
	CommandAborted=> , 
	Error=> , 
	ErrorID=> );
//凸轮表	
MC_CamTableSelect_Follower(
	Master:= ref_Master.Axis, 
	Slave:= ref_Follower.Axis, 
	CamTable:= CamTableFollower, 
	Execute:= ref_Follower.i.SelectCamTable, 
	Periodic:= TRUE, 
	MasterAbsolute:= , 
	SlaveAbsolute:= , 
	CamTableID:= iCamID, 
	Done=> ref_Follower.o.SelectCamTableDone, 
	Busy=> , 
	Error=> , 
	ErrorID=> );	
//凸轮位置	
MC_ReadCamTableSlaveDynamicsFollwer(
	Execute:= , 
	CamTableID:=iCamID , 
	MasterPosition:=ref_Master.o.ActPos , 
	Done=> , 
	Busy=> , 
	Error=> , 
	ErrorID=> , 
	SlavePosition=> , 
	SlaveVelocity=> , 
	SlaveAcceleration=> );
END_ACTION

ACTION CM02_Follower:
CASE FollowerSeq.Now OF
	0: 	   
	   IF Ref_MachineStateModel.Sts_Resetting  THEN
          FollowerSeq(ExeCute:=TRUE , Next:= Seq_Resetting);  
	   END_IF	
	
	   IF Ref_MachineStateModel.Sts_Stopping  THEN
		  FollowerSeq(ExeCute:=TRUE , Next:= Seq_Stopping);   
	   END_IF
	   IF Ref_MachineStateModel.Sts_Execute  THEN
		  FollowerSeq(ExeCute:= TRUE, Next:= 110);   
	   END_IF	   
{#region Resetting}	   
	Seq_Resetting:
		IF NOT ref_Follower.o.PowerOn  THEN;
		   ref_Follower.i.Enable:=TRUE;
		ELSE
		   FollowerSeq(ExeCute:=TRUE , Next:= 20); 
		END_IF
	    IF Ref_MachineStateModel.Sts_Stopping  THEN
		   FollowerSeq(ExeCute:= TRUE, Next:= Seq_Stopping);  
	    END_IF
		
	20:	
		IF NOT glb_AllAxisHomed_UN01 THEN
			FollowerSeq(ExeCute:=TRUE , Next:= 21);  
			ELSE
			FollowerSeq(ExeCute:=TRUE , Next:= 30); 
		END_IF
	   
	21:
	   iLastSeq:=0;
	   glb_lrBelt1WrkCnt:=0;
	   glb_lrBelt1TargetCnt:=0;
	   bRecipeComplete:=FALSE;
	   arDropBufferCyclinder[1].i.ActiveIn:=TRUE;
	   arDropBufferCyclinder[1].i.ActiveOut:=FALSE;
	   MEMSET(destAddr:= ADR(glb_BinBelt1), fillByte:= 0, n:= SIZEOF(glb_BinBelt1));   
	   FollowerSeq(ExeCute:=TRUE , Next:= 22); 
    22:
       tonFollowerSeq(IN:=TRUE , PT:=T#1S , Q=> , ET=> );
       IF tonFollowerSeq.Q AND arDropBufferCyclinder[1].i.InSensor THEN
		   tonFollowerSeq(IN:=FALSE , PT:=T#1S , Q=> , ET=> );
		   FollowerSeq(ExeCute:=TRUE , Next:= 23); 
       END_IF 
	   
	23:
	   ref_Follower.i.Home:=TRUE;
	   IF ref_Follower.o.HomeDone THEN
		   ref_Follower.i.Home:=FALSE;
		   FollowerSeq(ExeCute:=TRUE , Next:= 24); 
	   ELSE IF Ref_MachineStateModel.Sts_Stopping  THEN
		       ref_Follower.i.Home:=FALSE;
			   ref_Follower.i.Stop:=TRUE;
               FollowerSeq(ExeCute:=TRUE , Next:= Seq_Stopping);   
	        END_IF	   
	   END_IF	
	
    24: 
		
		FOR i:=1 TO 10 DO
			glb_BinBelt1.bin[1].arDrop[i]:=TRUE;	
	    END_FOR	
			glb_BinBelt1.bin[40].arDrop[40]:=TRUE;
	        glb_BinBelt1.bin[1].arDrop[HMI_B1DropBinNo]:=TRUE;
			lrPosCnt:=1;
			ref_Follower.i.Pos:=0;		
			FollowerSeq(ExeCute:=TRUE , Next:= 25);
		
	25:
        IF ref_Follower.o.StandStill THEN
		   FollowerSeq(Execute:= TRUE, Next:= 30);   
	    END_IF
		
    30:	//生产复位
	    ref_Follower.i.MoveAbs:=TRUE;
	    FollowerSeq(Execute:= TRUE, Next:= 31);   	
		
	31:
    	IF  ref_Follower.o.CmdDone THEN
		    ref_Follower.i.MoveAbs:=FALSE;
            FollowerSeq(Execute:= TRUE, Next:= Seq_ResettingDone);    	
		END_IF

   	Seq_ResettingDone: 
         IF NOT Ref_MachineStateModel.Sts_Resetting THEN
			FollowerSeq(ExeCute:=TRUE , Next:= 0); 	
		 END_IF	   
{end_Region}	
	 
    //自动运行
    110:
	    IF ilastSeq>100 THEN
		    FollowerSeq(ExeCute:=TRUE , Next:= ilastSeq);   
		ELSE 
			FollowerSeq(ExeCute:=TRUE , Next:= 111);  
		END_IF
	
	111:
		IF glb_lrBelt1WrkCnt < glb_lrBelt1TargetCnt THEN
			 FollowerSeq(ExeCute:=TRUE ,Hold:=FALSE, Next:= 120); 
		   ELSE IF glb_lrBelt1WrkCnt = glb_lrBelt1TargetCnt THEN
					FOR i:=1 TO 10 DO
						glb_BinBelt1.bin[1].arDrop[i]:=TRUE;
					END_FOR	
						glb_BinBelt1.bin[40].arDrop[40]:=TRUE;
						glb_BinBelt1.bin[1].arDrop[HMI_B1DropBinNo]:=TRUE;	
                        glb_lrBelt1WrkCnt:=0;
                        glb_lrBelt1TargetCnt:=0;	   
			    END_IF
		END_IF
	    IF Ref_MachineStateModel.Sts_Stopping  THEN
		   FollowerSeq(ExeCute:=TRUE , Next:= Seq_Stopping);   
	    END_IF
    120:  
	      FOR j:=1 TO 10 DO
			  IF  glb_BinBelt1.bin[j].arDrop[j] AND arCounters[j].Error THEN
				  glb_BinBelt1.bin[j].bReject:=TRUE;
			  END_IF			  
		  END_FOR

	      FOR j:=31 TO 40 DO
			  IF  glb_BinBelt1.bin[j].arDrop[j] AND arCounters[j].Error THEN
				  glb_BinBelt1.bin[j].bReject:=TRUE;
			  END_IF			  
		  END_FOR	
	
	      IF NOT glb_BinBelt1.bin[1].arDrop[1] AND NOT glb_BinBelt1.bin[2].arDrop[2] 
          AND NOT glb_BinBelt1.bin[3].arDrop[3] AND NOT glb_BinBelt1.bin[4].arDrop[4] 
          AND NOT glb_BinBelt1.bin[5].arDrop[5] AND NOT glb_BinBelt1.bin[6].arDrop[6]
          AND NOT glb_BinBelt1.bin[7].arDrop[7] AND NOT glb_BinBelt1.bin[8].arDrop[8] 
          AND NOT glb_BinBelt1.bin[9].arDrop[9] AND NOT glb_BinBelt1.bin[10].arDrop[10] 
		  AND NOT glb_BinBelt1.bin[31].arDrop[31] AND NOT glb_BinBelt1.bin[32].arDrop[32] 
          AND NOT glb_BinBelt1.bin[33].arDrop[33] AND NOT glb_BinBelt1.bin[34].arDrop[34]
          AND NOT glb_BinBelt1.bin[35].arDrop[35] AND NOT glb_BinBelt1.bin[36].arDrop[36]
          AND NOT glb_BinBelt1.bin[37].arDrop[37] AND NOT glb_BinBelt1.bin[38].arDrop[38] 
          AND NOT glb_BinBelt1.bin[39].arDrop[39] AND NOT glb_BinBelt1.bin[40].arDrop[40]
		  THEN
		      FollowerSeq(ExeCute:=TRUE ,Hold:=FALSE,Next:= 121);
          END_IF
		  IF Ref_MachineStateModel.Sts_Stopping  THEN
		     FollowerSeq(ExeCute:=TRUE , Next:= Seq_Stopping);   
	      END_IF
		  
    121: 		      
          IF NOT glb_BinBelt1.bin[HMI_B1DropBinNo].arDrop[HMI_B1DropBinNo] THEN
              FollowerSeq(ExeCute:=TRUE , Next:= 130); 	
		  ELSE  
			  FollowerSeq(ExeCute:=TRUE , Next:= 200); 	   
		  END_IF		  
	130:  
	      ref_Follower.i.Pos:=ref_Follower.i.Pos+215;
	      FollowerSeq(ExeCute:=TRUE ,Hold:=FALSE, Next:= 150);
	
	150:
	      ref_Follower.i.MoveAbs:=TRUE;
		  IF ref_Follower.o.CmdDone THEN
			 ref_Follower.i.MoveAbs:=FALSE;
			 FollowerSeq(ExeCute:=TRUE ,Hold:=FALSE, Next:= 300);
		  END_IF
	
	//往皮带3落料
	200:
	     IF glb_BinBelt3.bin[HMI_B3DropBinNo1].arDrop[HMI_B3DropBinNo1] THEN//皮带三对接工位
			FollowerSeq(ExeCute:=TRUE , Next:= 201); 	
		 END_IF
		 IF Ref_MachineStateModel.Sts_Stopping  THEN
		    FollowerSeq(ExeCute:=TRUE , Next:= Seq_Stopping);   
	     END_IF
		 
	201:
	     arDropBufferCyclinder[1].i.ActiveIn:=FALSE;
	     arDropBufferCyclinder[1].i.ActiveOut:=TRUE;
		 tonBufferCyclinderDelay(IN:= TRUE, PT:= T#500MS, Q=> , ET=> );
		 IF tonBufferCyclinderDelay.Q THEN
			tonBufferCyclinderDelay(IN:= FALSE, PT:= T#500MS, Q=> , ET=> );
			FollowerSeq(ExeCute:=TRUE ,Hold:=FALSE, Next:= 210);
		 END_IF
		 
		 
	210:
		  ref_Follower.i.Pos:=ref_Follower.i.Pos+215;
		  FollowerSeq(ExeCute:=TRUE ,Hold:=FALSE, Next:= 220);
	
	220:
	      ref_Follower.i.MoveAbs:=TRUE;
		  IF ref_Follower.o.CmdDone THEN
			 ref_Follower.i.MoveAbs:=FALSE;
			 FollowerSeq(ExeCute:=TRUE ,Hold:=FALSE, Next:= 221);
		  END_IF	
  
		  IF (ref_Follower.i.Pos-ref_Follower.o.ActPos) < 60 AND NOT bBeltInRange THEN
			  (*
		      glb_BinBelt3.bin[HMI_B3DropBinNo1].arDrop[HMI_B3DropBinNo1]:=FALSE;
			  glb_BinBelt3.bin[1].arDrop[HMI_B3DropBinNo2]:=TRUE;
		      glb_BinBelt3.bin[1].arDrop[HMI_B3DropBinNo3]:=TRUE; 
		      glb_BinBelt3.bin[HMI_B3DropBinNo1].Name:=glb_BinBelt1.bin[HMI_B1DropBinNo].Name;
		      glb_BinBelt3.bin[HMI_B3DropBinNo1].Amount:=glb_BinBelt1.bin[HMI_B1DropBinNo].Amount;			  
			  glb_lrBelt3ValidCnt:=glb_lrBelt3ValidCnt+1;
			  *)
			  bBeltInRange:=TRUE;
		  END_IF 
	  
	221:
	     arDropBufferCyclinder[1].i.ActiveIn:=TRUE;
	     arDropBufferCyclinder[1].i.ActiveOut:=FALSE;
		 IF arDropBufferCyclinder[1].i.InSensor AND NOT arDropBufferCyclinder[1].o.Error THEN
			FollowerSeq(ExeCute:=TRUE ,Hold:=FALSE, Next:= 230);
		 END_IF	
	
	
	230:
	      bBeltInRange:=FALSE;
		  glb_BinBelt3.bin[HMI_B3DropBinNo1].arDrop[HMI_B3DropBinNo1]:=FALSE;
		  glb_BinBelt3.bin[1].arDrop[HMI_B3DropBinNo2]:=TRUE;
		  glb_BinBelt3.bin[1].arDrop[HMI_B3DropBinNo3]:=TRUE; 
		  glb_BinBelt3.bin[HMI_B3DropBinNo1].Name:=glb_BinBelt1.bin[HMI_B1DropBinNo].Name;
		  glb_BinBelt3.bin[HMI_B3DropBinNo1].Amount:=glb_BinBelt1.bin[HMI_B1DropBinNo].Amount;			  
		  glb_lrBelt3ValidCnt:=glb_lrBelt3ValidCnt+1;		  
		  	  
		  glb_BinBelt1.bin[HMI_B1DropBinNo].arDrop[HMI_B1DropBinNo]:=FALSE;
		  FollowerSeq(ExeCute:=TRUE ,Hold:=FALSE, Next:= 300); 
		  
	300:
			glb_lrBelt1WrkCnt:=glb_lrBelt1WrkCnt+1;
			FOR i:=20 TO 1 BY -1 DO
				glb_BinBelt1.bin[i].arDrop:= glb_BinBelt1.bin[i-1].arDrop;
				glb_BinBelt1.bin[i].Amount:= glb_BinBelt1.bin[i-1].Amount;
				glb_BinBelt1.bin[i].Name:= glb_BinBelt1.bin[i-1].Name;
			END_FOR
			glb_BinBelt1.bin[31].arDrop[31]:=glb_BinBelt1.bin[10].arDrop[10];
			glb_BinBelt1.bin[32].arDrop[32]:=glb_BinBelt1.bin[9].arDrop[9];		     
			glb_BinBelt1.bin[33].arDrop[33]:=glb_BinBelt1.bin[8].arDrop[8];		
			glb_BinBelt1.bin[34].arDrop[34]:=glb_BinBelt1.bin[7].arDrop[7];
			glb_BinBelt1.bin[35].arDrop[35]:=glb_BinBelt1.bin[6].arDrop[6];
			glb_BinBelt1.bin[36].arDrop[36]:=glb_BinBelt1.bin[5].arDrop[5];
			glb_BinBelt1.bin[37].arDrop[37]:=glb_BinBelt1.bin[4].arDrop[4];
			glb_BinBelt1.bin[38].arDrop[38]:=glb_BinBelt1.bin[3].arDrop[3];
			glb_BinBelt1.bin[39].arDrop[39]:=glb_BinBelt1.bin[2].arDrop[2];	
			
			FollowerSeq(ExeCute:=TRUE ,Hold:=FALSE, Next:= 310); 
		  
	310:	  
			IF glb_lrBelt1WrkCnt < glb_lrBelt1TargetCnt-HMI_B1DropBinNo THEN
				 FollowerSeq(ExeCute:=TRUE ,Hold:=FALSE, Next:= 320); //数粒未完成
				 ELSE
				 FollowerSeq(ExeCute:=TRUE ,Hold:=FALSE, Next:= 400); //数粒已完成
			END_IF	
		  
	320:
			FOR i:=1 TO 10 DO
				glb_BinBelt1.bin[1].arDrop[i]:=TRUE;
			END_FOR	
			glb_BinBelt1.bin[40].arDrop[40]:=TRUE;
	        glb_BinBelt1.bin[1].arDrop[HMI_B1DropBinNo]:=TRUE;
	        FollowerSeq(ExeCute:=TRUE ,Hold:=FALSE, Next:= 111);
						
	
	400:
			FOR i:=1 TO 10 DO
				glb_BinBelt1.bin[1].arDrop[i]:=FALSE;
			END_FOR	
			glb_BinBelt1.bin[40].arDrop[40]:=FALSE;
	        glb_BinBelt1.bin[1].arDrop[HMI_B1DropBinNo]:=FALSE; 
            glb_BinBelt1.bin[1].Name:='END'; 	
			FollowerSeq(ExeCute:=TRUE ,Hold:=FALSE, Next:= 111);

		   
	
	Seq_Stopping:   
	    iLastSeq:= FollowerSeq.Last;
	    tonFollowerSeq(IN:=TRUE , PT:=T#1S , Q=> , ET=> );
		IF tonFollowerSeq.Q THEN
			tonFollowerSeq(IN:=FALSE , PT:=T#1S , Q=> , ET=> );
			FollowerSeq(ExeCute:=TRUE , Next:= Seq_StoppingDone); 
		END_IF
		

	Seq_StoppingDone:
	     ref_Follower.i.Disable:=TRUE;
		 IF NOT Ref_MachineStateModel.Sts_Stopping THEN
			FollowerSeq(ExeCute:=TRUE , Next:= 0); 
		 END_IF
END_CASE

FollowerSeq.Hold := Ref_MachineStateModel.Sts_Held;
END_ACTION

ACTION MainRoution:
EM_No:=2;
IF Ref_Unit.EM_Selected[EM_No] THEN
	IF Ref_MachineStateModel.Sts_Holding THEN
		Ref_Unit.EM_Holding_Done[EM_No]:=TRUE;
		ELSE
		Ref_Unit.EM_Holding_Done[EM_No]:=FALSE;
	END_IF
	IF Ref_MachineStateModel.Sts_UnHolding THEN
		Ref_Unit.EM_UnHolding_Done[EM_No]:=TRUE;
		ELSE
		Ref_Unit.EM_UnHolding_Done[EM_No]:=FALSE;
	END_IF
	
	IF Ref_MachineStateModel.Sts_Suspending THEN
		Ref_Unit.EM_Suspending_Done[EM_No]:=TRUE;
		ELSE
		Ref_Unit.EM_Suspending_Done[EM_No]:=FALSE;
	END_IF
	
	IF Ref_MachineStateModel.Sts_UnSuspending THEN
		Ref_Unit.EM_UnSuspending_Done[EM_No]:=TRUE;
		ELSE
		Ref_Unit.EM_UnSuspending_Done[EM_No]:=FALSE;
	END_IF
	
	IF Ref_MachineStateModel.Sts_Resetting  AND FollowerSeq.Now=Seq_ResettingDone THEN
	   Ref_Unit.EM_Resetting_Done[EM_No]:=TRUE;
       ELSE   
	   Ref_Unit.EM_Resetting_Done[EM_No]:=FALSE;
	END_IF
	
	IF Ref_MachineStateModel.Sts_Clearing THEN
	   Ref_Unit.EM_Clearing_Done[EM_No]:=TRUE;
	   ELSE
	   Ref_Unit.EM_Clearing_Done[EM_No]:=FALSE;
	END_IF
	

	IF Ref_MachineStateModel.Sts_Starting THEN
	   Ref_Unit.EM_Starting_Done[EM_No]:=TRUE;
	   ELSE
       Ref_Unit.EM_Starting_Done[EM_No]:=FALSE;
	END_IF
	
	IF Ref_MachineStateModel.Sts_Stopping AND FollowerSeq.Now=Seq_StoppingDone  THEN
	   Ref_Unit.EM_Stopping_Done[EM_No]:=TRUE;	
       ELSE  
	   Ref_Unit.EM_Stopping_Done[EM_No]:=FALSE;	
	END_IF

	IF Ref_MachineStateModel.Sts_Aborting THEN
	    FollowerSeq(ExeCute:=TRUE , Next:= 0); 		
		IF ref_Follower.o.InSync THEN	 
		   ref_Follower.i.CamOut:=TRUE;
		ELSE IF  NOT ref_Follower.o.StandStill THEN
				ref_follower.i.Stop:=TRUE;
			END_IF
		END_IF  
	
		IF tonAbortingWatchDog.Q THEN 
			Ref_Unit.EM_Aborting_Done[EM_No]:=TRUE;
			ref_Follower.i.Disable:=TRUE;
        END_IF
    ELSE
		Ref_Unit.EM_Aborting_Done[EM_No]:=FALSE;
	END_IF
	
	tonAbortingWatchDog(IN:= Ref_MachineStateModel.Sts_Aborting, PT:=T#3S , Q=> , ET=> );
	CM02_Follower();
ELSE
FollowerSeq(ExeCute:=TRUE , Next:= 0); 	
		
END_IF
END_ACTION

ACTION SR999_FaultHandler:
;
END_ACTION

END_PROGRAM

// ---- POUs/PackMaL_UN01/EM03_Follower2.TcPOU
PROGRAM EM03_Follower2
VAR
	ref_Master: REFERENCE TO UDT_AXISADMIN;
	ref_Follower: REFERENCE TO UDT_AXISADMIN;
	Ref_MachineStateModel: REFERENCE TO PackMlv3_StateModel;
	Ref_Unit: REFERENCE TO UDT_UnitAdmin;
	EM_No: INT:=3;
	tonAbortingWatchDog: TON;
	tonStoppingWatchDog: Ton;
	MC_CamIn_Follower: MC_CamIn;

	MC_CamTableSelect_Follower: MC_CamTableSelect;
	CamTableFollower: MC_CAM_REF;
	table1: ARRAY[1..2] OF MC_MotionFunctionPoint; (*用于定义电子凸轮表中的关键点*)


    MC_ReadCamTableSlaveDynamicsFollwer: MC_ReadCamTableSlaveDynamics;
	
	tonFollowerSeq: TON;
	FollowerSeq: SequenceTransfer;	
	
	i: INT;
	lrPosCnt: LREAL;
	bRecipeComplete: BOOL;
	bBeltInRange: BOOL;
	iLastSeq: INT;
	j: INT;
	tonBufferCyclinderDelay: TON;
END_VAR

VAR CONSTANT
	iCamID: MC_CAM_ID:=2;		
END_VAR

//减速比10/1 同步轮周长400 ，皮带总长5200，26个工位，工位间距200
Ref_MachineStateModel REF= UN01_MachineStateModel;
Ref_Unit REF=Unit01;
ref_Master REF= arVirtualAxisAdmin[1];
ref_Follower REF= arRealAxisAdmin[42];
MainRoution();
CM01_Cam();
SR999_Faulthandler();

ACTION CM01_Cam:
//凸轮1曲线
camTableFollower.ArraySize:=SIZEOF(table1);
camTableFollower.NoOfColumns:=1;
camTableFollower.NoOfRows:=2;
camTableFollower.pArray:=ADR(table1);
camTableFollower.TableType:=MC_TABLETYPE_MOTIONFUNCTION;

table1[1].FunctionType:=MOTIONFUNCTYPE_POLYNOM1;
table1[1].MasterPos:=0;
table1[1].SlavePos:=0;
table1[1].PointIndex:=1;
table1[1].PointType:=MOTIONPOINTTYPE_MOTION;
		
table1[2].FunctionType:=MOTIONFUNCTYPE_POLYNOM1;
table1[2].MasterPos:=200;
table1[2].SlavePos:=200;
table1[2].PointIndex:=2;
table1[2].PointType:=MOTIONPOINTTYPE_MOTION;

MC_CamIn_Follower(
	Master:= ref_Master.Axis, 
	Slave:= ref_Follower.Axis, 
	Execute:= ref_Follower.i.CamIn, 
	MasterOffset:= , 
	SlaveOffset:= , 
	MasterScaling:= 1, 
	SlaveScaling:= 1, 
	StartMode:= MC_STARTMODE_ABSOLUTE, 
	CamTableID:= iCamID, 
	BufferMode:= , 
	Options:= , 
	InSync=> , 
	Busy=> , 
	Active=> , 
	CommandAborted=> , 
	Error=> , 
	ErrorID=> );
	
MC_CamTableSelect_Follower(
	Master:= ref_Master.Axis, 
	Slave:= ref_Follower.Axis, 
	CamTable:= CamTableFollower, 
	Execute:= ref_Follower.i.SelectCamTable, 
	Periodic:= TRUE, 
	MasterAbsolute:= , 
	SlaveAbsolute:= , 
	CamTableID:= iCamID, 
	Done=> ref_Follower.o.SelectCamTableDone, 
	Busy=> , 
	Error=> , 
	ErrorID=> );	
	
MC_ReadCamTableSlaveDynamicsFollwer(
	Execute:= , 
	CamTableID:=iCamID , 
	MasterPosition:=ref_Master.o.ActPos , 
	Done=> , 
	Busy=> , 
	Error=> , 
	ErrorID=> , 
	SlavePosition=> , 
	SlaveVelocity=> , 
	SlaveAcceleration=> );
END_ACTION

ACTION CM02_Follower:
CASE FollowerSeq.Now OF
	0: 	   
	   IF Ref_MachineStateModel.Sts_Resetting  THEN
          FollowerSeq(ExeCute:=TRUE , Next:= Seq_Resetting);  
	   END_IF	
	
	   IF Ref_MachineStateModel.Sts_Stopping  THEN
		  FollowerSeq(ExeCute:=TRUE , Next:= Seq_Stopping);   
	   END_IF
	   IF Ref_MachineStateModel.Sts_Execute  THEN
		  FollowerSeq(ExeCute:= TRUE, Next:= 110);   
	   END_IF	   
{#region Resetting}	   
	Seq_Resetting:
		IF NOT ref_Follower.o.PowerOn  THEN;
		   ref_Follower.i.Enable:=TRUE;
		ELSE
		   FollowerSeq(ExeCute:=TRUE , Next:= 20); 
		END_IF
	    IF Ref_MachineStateModel.Sts_Stopping  THEN
		   FollowerSeq(ExeCute:= TRUE, Next:= Seq_Stopping);  
	    END_IF
		
	20:	
		IF NOT glb_AllAxisHomed_UN01 THEN
			FollowerSeq(ExeCute:=TRUE , Next:= 21);  
			ELSE
			FollowerSeq(ExeCute:=TRUE , Next:= 30); 
		END_IF
	   
	21:
	   iLastSeq:=0;
	   glb_lrBelt2TargetCnt:=0;
       glb_lrBelt2WrkCnt:=0;
	   bRecipeComplete:=FALSE;
	   arDropBufferCyclinder[2].i.ActiveIn:=TRUE;
	   arDropBufferCyclinder[2].i.ActiveOut:=FALSE;
	   
       MEMSET(destAddr:= ADR(glb_BinBelt2), fillByte:= 0, n:= SIZEOF(glb_BinBelt2));    
	   FollowerSeq(ExeCute:=TRUE , Next:= 22); 
	   
    22:
       tonFollowerSeq(IN:=TRUE , PT:=T#1S , Q=> , ET=> );
       IF tonFollowerSeq.Q AND arDropBufferCyclinder[2].i.InSensor THEN
		   tonFollowerSeq(IN:=FALSE , PT:=T#1S , Q=> , ET=> );
		   FollowerSeq(ExeCute:=TRUE , Next:= 23); 
       END_IF 
	23:
	   ref_Follower.i.Home:=TRUE;
	   IF ref_Follower.o.HomeDone THEN
		   ref_Follower.i.Home:=FALSE;
		   FollowerSeq(ExeCute:=TRUE , Next:= 24); 
	   ELSE IF Ref_MachineStateModel.Sts_Stopping  THEN
		       ref_Follower.i.Home:=FALSE;
			   ref_Follower.i.stop:=TRUE;
               FollowerSeq(ExeCute:=TRUE , Next:= Seq_Stopping);   
	        END_IF	   
	   END_IF	
	   
    24: 
		FOR i:=1 TO 10 DO
			glb_BinBelt2.bin[1].arDrop[i]:=TRUE;
	    END_FOR			
			glb_BinBelt2.bin[1].arDrop[HMI_B2DropBinNo]:=TRUE;
			glb_BinBelt2.bin[40].arDrop[40]:=TRUE;
        lrPosCnt:=1;
		ref_Follower.i.Pos:=0;		
		FollowerSeq(ExeCute:=TRUE , Next:= 25);
		
	25:
        IF ref_Follower.o.StandStill THEN
		   FollowerSeq(Execute:= TRUE, Next:= 30);   
	    END_IF
		
    30:	//生产复位
	    ref_Follower.i.MoveAbs:=TRUE;
	    FollowerSeq(Execute:= TRUE, Next:= 31);   	
		
	31:
    	IF  ref_Follower.o.CmdDone THEN
		    ref_Follower.i.MoveAbs:=FALSE;
            FollowerSeq(Execute:= TRUE, Next:= Seq_ResettingDone);    	
		END_IF

   	Seq_ResettingDone: 
         IF NOT Ref_MachineStateModel.Sts_Resetting THEN
			FollowerSeq(ExeCute:=TRUE , Next:= 0); 	
		 END_IF	   
{end_region}
	
    //自动运行
    110:	
	     IF iLastSeq>100 THEN
			 FollowerSeq(ExeCute:=TRUE , Next:= iLastSeq);
		 ELSE 
	         FollowerSeq(ExeCute:=TRUE , Next:= 111);
		 END_IF
	
	111:
		  IF glb_lrBelt2WrkCnt < glb_lrBelt2TargetCnt THEN
			 FollowerSeq(ExeCute:=TRUE ,Hold:=FALSE, Next:= 120);
		  ELSE IF glb_lrBelt2WrkCnt = glb_lrBelt2TargetCnt THEN
					FOR i:=1 TO 10 DO
						glb_BinBelt2.bin[1].arDrop[i]:=TRUE;
					END_FOR	
						glb_BinBelt2.bin[1].arDrop[HMI_B2DropBinNo]:=TRUE;
			    		glb_BinBelt2.bin[40].arDrop[40]:=TRUE;	
                   glb_lrBelt2WrkCnt:=0;
                   glb_lrBelt2TargetCnt:=0;	 
			   END_IF
		  END_IF  
		  IF Ref_MachineStateModel.Sts_Stopping  THEN
		     FollowerSeq(ExeCute:=TRUE , Next:= Seq_Stopping);   
	      END_IF		  
    120:  
	
		  FOR j:=1 TO 10 DO
			  IF  glb_BinBelt2.bin[j].arDrop[j] AND arCounters[j].Error THEN
				  glb_BinBelt2.bin[j].bReject:=TRUE;
			  END_IF			  
		  END_FOR

	      FOR j:=31 TO 40 DO
			  IF  glb_BinBelt2.bin[j].arDrop[j] AND arCounters[j].Error THEN
				  glb_BinBelt2.bin[j].bReject:=TRUE;
			  END_IF			  
		  END_FOR	
	
	      IF NOT glb_BinBelt2.bin[1].arDrop[1] 
          AND NOT glb_BinBelt2.bin[2].arDrop[2] 
          AND NOT glb_BinBelt2.bin[3].arDrop[3] 
          AND NOT glb_BinBelt2.bin[4].arDrop[4] 
          AND NOT glb_BinBelt2.bin[5].arDrop[5] 
          AND NOT glb_BinBelt2.bin[6].arDrop[6]
          AND NOT glb_BinBelt2.bin[7].arDrop[7] 
          AND NOT glb_BinBelt2.bin[8].arDrop[8] 
          AND NOT glb_BinBelt2.bin[9].arDrop[9] 
          AND NOT glb_BinBelt2.bin[10].arDrop[10] 
		  AND NOT glb_BinBelt2.bin[31].arDrop[31] 
          AND NOT glb_BinBelt2.bin[32].arDrop[32] 
          AND NOT glb_BinBelt2.bin[33].arDrop[33] 
          AND NOT glb_BinBelt2.bin[34].arDrop[34] 
          AND NOT glb_BinBelt2.bin[35].arDrop[35] 
          AND NOT glb_BinBelt2.bin[36].arDrop[36]
          AND NOT glb_BinBelt2.bin[37].arDrop[37] 
          AND NOT glb_BinBelt2.bin[38].arDrop[38] 
          AND NOT glb_BinBelt2.bin[39].arDrop[39] 
          AND NOT glb_BinBelt2.bin[40].arDrop[40] THEN
              FollowerSeq(ExeCute:=TRUE ,Hold:=FALSE, Next:= 121); 
          END_IF
		  
		  IF Ref_MachineStateModel.Sts_Stopping  THEN
		     FollowerSeq(ExeCute:=TRUE , Next:= Seq_Stopping);   
	      END_IF
	121:  	
          IF NOT glb_BinBelt2.bin[HMI_B2DropBinNo].arDrop[HMI_B2DropBinNo] THEN 
              FollowerSeq(ExeCute:=TRUE , Next:= 130); 	
		  ELSE  //落料到皮带3	  
			  FollowerSeq(ExeCute:=TRUE , Next:= 200); 	
		  END_IF
		  
	130:  
	      ref_Follower.i.Pos:=ref_Follower.i.Pos+215;
	      FollowerSeq(ExeCute:=TRUE ,Hold:=FALSE, Next:= 150);
	
	150:
	      ref_Follower.i.MoveAbs:=TRUE;
		  IF ref_Follower.o.CmdDone THEN
			 ref_Follower.i.MoveAbs:=FALSE;
			 FollowerSeq(ExeCute:=TRUE ,Hold:=FALSE, Next:= 300);
		  END_IF
	

	200://等待皮带3信号
		IF glb_BinBelt3.bin[HMI_B3DropBinNo2].arDrop[HMI_B3DropBinNo2] THEN
			FollowerSeq(ExeCute:=TRUE , Next:= 201); 
		END_IF
		IF Ref_MachineStateModel.Sts_Stopping  THEN
			FollowerSeq(ExeCute:=TRUE , Next:= Seq_Stopping);   
		END_IF	
	201:
	     arDropBufferCyclinder[2].i.ActiveIn:=FALSE;
	     arDropBufferCyclinder[2].i.ActiveOut:=TRUE;
		 tonBufferCyclinderDelay(IN:= TRUE, PT:= T#500MS, Q=> , ET=> );
		 IF tonBufferCyclinderDelay.Q THEN
			tonBufferCyclinderDelay(IN:= FALSE, PT:= T#500MS, Q=> , ET=> );
			FollowerSeq(ExeCute:=TRUE ,Hold:=FALSE, Next:= 210);
		 END_IF		
	210:
		  ref_Follower.i.Pos:=ref_Follower.i.Pos+215;
		  FollowerSeq(ExeCute:=TRUE ,Hold:=FALSE, Next:= 220);
	
	220:
	      ref_Follower.i.MoveAbs:=TRUE;
		  IF ref_Follower.o.CmdDone THEN
			 ref_Follower.i.MoveAbs:=FALSE;
			 FollowerSeq(ExeCute:=TRUE ,Hold:=FALSE, Next:= 221);
		  END_IF
		  IF (ref_Follower.i.Pos-ref_Follower.o.ActPos) < 60 AND NOT bBeltInRange THEN
		   //   glb_BinBelt3.bin[HMI_B3DropBinNo2].arDrop[HMI_B3DropBinNo2]:=FALSE;
			  bBeltInRange:=TRUE;
		  END_IF 
		  
	221:
	     arDropBufferCyclinder[2].i.ActiveIn:=TRUE;
	     arDropBufferCyclinder[2].i.ActiveOut:=FALSE;
		 IF arDropBufferCyclinder[2].i.InSensor AND NOT arDropBufferCyclinder[2].o.Error THEN
			FollowerSeq(ExeCute:=TRUE ,Hold:=FALSE, Next:= 230);
		 END_IF	  	
	
		 
	230:
	      bBeltInRange:=FALSE;
		  glb_BinBelt3.bin[HMI_B3DropBinNo2].arDrop[HMI_B3DropBinNo2]:=FALSE;
		  glb_BinBelt2.bin[HMI_B2DropBinNo].arDrop[HMI_B2DropBinNo]:=FALSE;
		  FollowerSeq(ExeCute:=TRUE ,Hold:=FALSE, Next:= 300); 
		  
	300:
	     glb_lrBelt2WrkCnt:=glb_lrBelt2WrkCnt+1;
	      FOR i:=20 TO 1 BY -1 DO
			  glb_BinBelt2.bin[i].arDrop:= glb_BinBelt2.bin[i-1].arDrop;
		  END_FOR
			glb_BinBelt2.bin[31].arDrop[31]:=glb_BinBelt2.bin[10].arDrop[10];
			glb_BinBelt2.bin[32].arDrop[32]:=glb_BinBelt2.bin[9].arDrop[9];		     
			glb_BinBelt2.bin[33].arDrop[33]:=glb_BinBelt2.bin[8].arDrop[8];		
			glb_BinBelt2.bin[34].arDrop[34]:=glb_BinBelt2.bin[7].arDrop[7];
			glb_BinBelt2.bin[35].arDrop[35]:=glb_BinBelt2.bin[6].arDrop[6];
			glb_BinBelt2.bin[36].arDrop[36]:=glb_BinBelt2.bin[5].arDrop[5];
			glb_BinBelt2.bin[37].arDrop[37]:=glb_BinBelt2.bin[4].arDrop[4];
			glb_BinBelt2.bin[38].arDrop[38]:=glb_BinBelt2.bin[3].arDrop[3];
			glb_BinBelt2.bin[39].arDrop[39]:=glb_BinBelt2.bin[2].arDrop[2];			  
			FollowerSeq(ExeCute:=TRUE ,Hold:=FALSE, Next:= 310); 
		  	  
		  
	310:	  
	      IF glb_lrBelt2WrkCnt < glb_lrBelt2TargetCnt-HMI_B2DropBinNo THEN
			 FollowerSeq(ExeCute:=TRUE , Next:= 320); //数粒未完成
             ELSE
	         FollowerSeq(ExeCute:=TRUE , Next:= 400); //数粒已完成
		  END_IF	
	320:
			FOR i:=1 TO 10 DO
				glb_BinBelt2.bin[1].arDrop[i]:=TRUE;
			END_FOR	
				glb_BinBelt2.bin[1].arDrop[HMI_B2DropBinNo]:=TRUE;
			    glb_BinBelt2.bin[40].arDrop[40]:=TRUE;
	        FollowerSeq(ExeCute:=TRUE ,Hold:=FALSE, Next:= 111);
	
	400://数粒已完成
			FOR i:=1 TO 10 DO
				glb_BinBelt2.bin[1].arDrop[i]:=FALSE;
			END_FOR	
				glb_BinBelt2.bin[1].arDrop[HMI_B2DropBinNo]:=FALSE;
			    glb_BinBelt2.bin[40].arDrop[40]:=FALSE;
			FollowerSeq(ExeCute:=TRUE ,Hold:=FALSE, Next:= 111);
			

		  
	Seq_Stopping:   
	    iLastSeq:= FollowerSeq.Last;
	    tonFollowerSeq(IN:=TRUE , PT:=T#1S , Q=> , ET=> );
		IF tonFollowerSeq.Q THEN
			tonFollowerSeq(IN:=FALSE , PT:=T#1S , Q=> , ET=> );
			FollowerSeq(ExeCute:=TRUE , Next:= Seq_StoppingDone); 
		END_IF
		

	Seq_StoppingDone:
	     ref_Follower.i.Disable:=TRUE;
		 IF NOT Ref_MachineStateModel.Sts_Stopping THEN
			FollowerSeq(ExeCute:=TRUE , Next:= 0); 
		 END_IF
END_CASE
FollowerSeq.Hold := Ref_MachineStateModel.Sts_Held;
END_ACTION

ACTION MainRoution:
EM_No:=3;
IF Ref_Unit.EM_Selected[EM_No] THEN
	IF Ref_MachineStateModel.Sts_Holding THEN
		Ref_Unit.EM_Holding_Done[EM_No]:=TRUE;
		ELSE
		Ref_Unit.EM_Holding_Done[EM_No]:=FALSE;
	END_IF
	IF Ref_MachineStateModel.Sts_UnHolding THEN
		Ref_Unit.EM_UnHolding_Done[EM_No]:=TRUE;
		ELSE
		Ref_Unit.EM_UnHolding_Done[EM_No]:=FALSE;
	END_IF
	
	IF Ref_MachineStateModel.Sts_Suspending THEN
		Ref_Unit.EM_Suspending_Done[EM_No]:=TRUE;
		ELSE
		Ref_Unit.EM_Suspending_Done[EM_No]:=FALSE;
	END_IF
	
	IF Ref_MachineStateModel.Sts_UnSuspending THEN
		Ref_Unit.EM_UnSuspending_Done[EM_No]:=TRUE;
		ELSE
		Ref_Unit.EM_UnSuspending_Done[EM_No]:=FALSE;
	END_IF
	
	IF Ref_MachineStateModel.Sts_Resetting  AND FollowerSeq.Now=Seq_ResettingDone THEN
	   Ref_Unit.EM_Resetting_Done[EM_No]:=TRUE;
       ELSE   
	   Ref_Unit.EM_Resetting_Done[EM_No]:=FALSE;
	END_IF
	
	IF Ref_MachineStateModel.Sts_Clearing THEN
	   Ref_Unit.EM_Clearing_Done[EM_No]:=TRUE;
	   ELSE
	   Ref_Unit.EM_Clearing_Done[EM_No]:=FALSE;
	END_IF
	

	IF Ref_MachineStateModel.Sts_Starting THEN
	   Ref_Unit.EM_Starting_Done[EM_No]:=TRUE;
	   ELSE
       Ref_Unit.EM_Starting_Done[EM_No]:=FALSE;
	END_IF
	
	IF Ref_MachineStateModel.Sts_Stopping AND FollowerSeq.Next=Seq_StoppingDone  THEN
	   Ref_Unit.EM_Stopping_Done[EM_No]:=TRUE;	
       ELSE  
	   Ref_Unit.EM_Stopping_Done[EM_No]:=FALSE;	
	END_IF

	IF Ref_MachineStateModel.Sts_Aborting THEN
		
       FollowerSeq(ExeCute:=TRUE , Next:= 0);
		IF ref_Follower.o.InSync THEN	 
		   ref_Follower.i.CamOut:=TRUE;
		ELSE IF  NOT ref_Follower.o.StandStill THEN
				ref_follower.i.Stop:=TRUE;
			END_IF
		END_IF  	
				
		IF tonAbortingWatchDog.Q THEN 
			Ref_Unit.EM_Aborting_Done[EM_No]:=TRUE;
			ref_Follower.i.Disable:=TRUE;
        END_IF
    ELSE
		Ref_Unit.EM_Aborting_Done[EM_No]:=FALSE;
	END_IF
	
	tonAbortingWatchDog(IN:= Ref_MachineStateModel.Sts_Aborting, PT:=T#3S , Q=> , ET=> );
	CM02_Follower();
ELSE
FollowerSeq(ExeCute:=TRUE , Next:= 0); 			
END_IF
END_ACTION

ACTION SR999_FaultHandler:
;
END_ACTION

END_PROGRAM

// ---- POUs/PackMaL_UN01/EM04_Follower3.TcPOU
PROGRAM EM04_Follower3
VAR
	ref_Master: REFERENCE TO UDT_AXISADMIN;
	ref_Follower: REFERENCE TO UDT_AXISADMIN;
	Ref_MachineStateModel: REFERENCE TO PackMlv3_StateModel;
	Ref_Unit: REFERENCE TO UDT_UnitAdmin;
	EM_No: INT:=4;
	tonAbortingWatchDog: TON;
	tonStoppingWatchDog: Ton;
	MC_CamIn_Follower: MC_CamIn;

	MC_CamTableSelect_Follower: MC_CamTableSelect;
	CamTableFollower: MC_CAM_REF;
	table1: ARRAY[1..2] OF MC_MotionFunctionPoint; (*用于定义电子凸轮表中的关键点*)


    MC_ReadCamTableSlaveDynamicsFollwer: MC_ReadCamTableSlaveDynamics;
	
	tonFollowerSeq: TON;
	FollowerSeq: SequenceTransfer;	
	
	i: INT;
	lrPosCnt: INT;
	bRecipeComplete: BOOL;
	bBeltInRange: BOOL;
	iLastSeq: INT;
END_VAR

VAR CONSTANT
	iCamID: MC_CAM_ID:=3;		
END_VAR

(*减速比10/1 同步轮周长400 ，皮带总长11600，58个工位，工位间距200
28个工位后开始落料*)
Ref_MachineStateModel REF= UN01_MachineStateModel;
Ref_Unit REF=Unit01;
ref_Master REF= arVirtualAxisAdmin[1];
ref_Follower REF= arRealAxisAdmin[43];
MainRoution();
CM01_Cam();
SR999_Faulthandler();

ACTION CM01_Cam:
//凸轮1曲线
camTableFollower.ArraySize:=SIZEOF(table1);
camTableFollower.NoOfColumns:=1;
camTableFollower.NoOfRows:=2;
camTableFollower.pArray:=ADR(table1);
camTableFollower.TableType:=MC_TABLETYPE_MOTIONFUNCTION;

table1[1].FunctionType:=MOTIONFUNCTYPE_POLYNOM1;
table1[1].MasterPos:=0;
table1[1].SlavePos:=0;
table1[1].PointIndex:=1;
table1[1].PointType:=MOTIONPOINTTYPE_MOTION;
		
table1[2].FunctionType:=MOTIONFUNCTYPE_POLYNOM1;
table1[2].MasterPos:=200;
table1[2].SlavePos:=200;
table1[2].PointIndex:=2;
table1[2].PointType:=MOTIONPOINTTYPE_MOTION;

MC_CamIn_Follower(
	Master:= ref_Master.Axis, 
	Slave:= ref_Follower.Axis, 
	Execute:= ref_Follower.i.CamIn , 
	MasterOffset:= , 
	SlaveOffset:= , 
	MasterScaling:= 1, 
	SlaveScaling:= 1, 
	StartMode:= MC_STARTMODE_ABSOLUTE, 
	CamTableID:= iCamID, 
	BufferMode:= , 
	Options:= , 
	InSync=> , 
	Busy=> , 
	Active=> , 
	CommandAborted=> , 
	Error=> , 
	ErrorID=> );
	
MC_CamTableSelect_Follower(
	Master:= ref_Master.Axis, 
	Slave:= ref_Follower.Axis, 
	CamTable:= CamTableFollower, 
	Execute:= ref_Follower.i.SelectCamTable , 
	Periodic:= TRUE, 
	MasterAbsolute:= , 
	SlaveAbsolute:= , 
	CamTableID:= iCamID, 
	Done=> ref_Follower.o.SelectCamTableDone, 
	Busy=> , 
	Error=> , 
	ErrorID=> );	
	
MC_ReadCamTableSlaveDynamicsFollwer(
	Execute:= , 
	CamTableID:=iCamID , 
	MasterPosition:=ref_Master.o.ActPos, 
	Done=> , 
	Busy=> , 
	Error=> , 
	ErrorID=> , 
	SlavePosition=> , 
	SlaveVelocity=> , 
	SlaveAcceleration=> );
END_ACTION

ACTION CM02_Follower:
CASE FollowerSeq.Now OF
	0: 	   
	   IF Ref_MachineStateModel.Sts_Resetting  THEN
          FollowerSeq(ExeCute:=TRUE , Next:= Seq_Resetting);  
	   END_IF	
	
	   IF Ref_MachineStateModel.Sts_Stopping  THEN
		  FollowerSeq(ExeCute:=TRUE , Next:= Seq_Stopping);   
	   END_IF
	   IF Ref_MachineStateModel.Sts_Execute  THEN
		  FollowerSeq(ExeCute:= TRUE, Next:= 110);   
	   END_IF	   
{#region resetting}	   
	Seq_Resetting:
		IF NOT ref_Follower.o.PowerOn  THEN;
		   ref_Follower.i.Enable:=TRUE;
		ELSE
		   FollowerSeq(ExeCute:=TRUE , Next:= 20); 
		END_IF
	    IF Ref_MachineStateModel.Sts_Stopping  THEN
		   FollowerSeq(ExeCute:= TRUE, Next:= Seq_Stopping);  
	    END_IF
		
	20:	
		IF NOT glb_AllAxisHomed_UN01 THEN
			FollowerSeq(ExeCute:=TRUE , Next:= 21);  
			ELSE
			FollowerSeq(ExeCute:=TRUE , Next:= 30); 
		END_IF
	   
	21:
	   iLastSeq:=0;
	   glb_lrBelt3TargetCnt:=0;
	   glb_lrBelt3WrkCnt:=0;
	   glb_lrBelt3ValidCnt:=0;
	   bRecipeComplete:=FALSE;
	   arDropBufferCyclinder[1].i.ActiveIn:=TRUE;
	   arDropBufferCyclinder[1].i.ActiveOut:=FALSE;
	   MEMSET(destAddr:= ADR(glb_BinBelt3), fillByte:= 0, n:= SIZEOF(glb_BinBelt3));      
	   FollowerSeq(ExeCute:=TRUE , Next:= 22); 
	22:
       tonFollowerSeq(IN:=TRUE , PT:=T#1S , Q=> , ET=> );
       IF tonFollowerSeq.Q AND arDropBufferCyclinder[1].I.InSensor 
       AND arDropBufferCyclinder[2].i.InSensor THEN
		   tonFollowerSeq(IN:=FALSE , PT:=T#1S , Q=> , ET=> );
		   FollowerSeq(ExeCute:=TRUE , Next:= 23); 
       END_IF 
	   
	23:
	   ref_Follower.i.Home:=TRUE;
	   IF ref_Follower.o.HomeDone THEN
		   ref_Follower.i.Home:=FALSE;
		   FollowerSeq(ExeCute:=TRUE , Next:= 24); 
	   ELSE IF Ref_MachineStateModel.Sts_Stopping  THEN
		       ref_Follower.i.Home:=FALSE;
			   ref_Follower.i.Stop:=TRUE;
               FollowerSeq(ExeCute:=TRUE , Next:= Seq_Stopping);   
	        END_IF	   
	   END_IF	
		
    24: 
		glb_BinBelt3.bin[1].arDrop[HMI_B3DropBinNo1]:=TRUE;
		glb_BinBelt3.bin[1].arDrop[HMI_B3DropBinNo2]:=TRUE;
		glb_BinBelt3.bin[1].arDrop[HMI_B3DropBinNo3]:=TRUE;
        lrPosCnt:=1;
		ref_Follower.i.Pos:=0;		
		FollowerSeq(ExeCute:=TRUE , Next:= 25);
		
	25:
        IF ref_Follower.o.StandStill THEN
		   FollowerSeq(Execute:= TRUE, Next:= 30);   
	    END_IF
		
    30:	//生产复位
	    ref_Follower.i.MoveAbs:=TRUE; 	
    	IF  ref_Follower.o.CmdDone THEN
		    ref_Follower.i.MoveAbs:=FALSE;
            FollowerSeq(Execute:= TRUE, Next:= Seq_ResettingDone);    	
		END_IF

		
   	Seq_ResettingDone: 
         IF NOT Ref_MachineStateModel.Sts_Resetting THEN
			FollowerSeq(ExeCute:=TRUE , Next:= 0); 	
		 END_IF	   
{end_region}
	
    //自动运行
    110:
        IF iLastSeq>100 THEN
	       FollowerSeq(ExeCute:=TRUE , Next:= iLastSeq);
        ELSE 
		   FollowerSeq(ExeCute:=TRUE , Next:= 111);
		END_IF
    111: 
        IF glb_BinBelt1.bin[HMI_B1DropBinNo].arDrop[HMI_B1DropBinNo] THEN //等待皮带1倒药
		   FollowerSeq(ExeCute:=TRUE , Next:= 112);
		END_IF
		
		IF NOT glb_BinBelt1.bin[HMI_B1DropBinNo].arDrop[HMI_B1DropBinNo] 
		   AND glb_lrBelt3ValidCnt > 0  THEN // AND glb_lrBelt1WrkCnt=0 
			FollowerSeq(ExeCute:=TRUE , Next:= 120);
		END_IF
		
		IF Ref_MachineStateModel.Sts_Stopping  THEN
			FollowerSeq(ExeCute:=TRUE , Next:= Seq_Stopping);   
		END_IF   		
    112:
		   glb_BinBelt3.bin[1].arDrop[HMI_B3DropBinNo1]:=TRUE;
//		   glb_BinBelt3.bin[1].arDrop[HMI_B3DropBinNo2]:=FALSE;
//		   glb_BinBelt3.bin[1].arDrop[HMI_B3DropBinNo3]:=FALSE; 
           FollowerSeq(ExeCute:=TRUE , Next:= 120); 	
    120:  
	      IF NOT glb_BinBelt3.bin[HMI_B3DropBinNo1].arDrop[HMI_B3DropBinNo1] 
          AND NOT glb_BinBelt3.bin[HMI_B3DropBinNo2].arDrop[HMI_B3DropBinNo2] THEN 
              FollowerSeq(ExeCute:=TRUE , Next:= 121); 	
		  END_IF
		  IF Ref_MachineStateModel.Sts_Stopping  THEN
		     FollowerSeq(ExeCute:=TRUE , Next:= Seq_Stopping);   
	      END_IF
		  
    121: 
         IF NOT glb_BinBelt3.bin[HMI_B3DropBinNo3].arDrop[HMI_B3DropBinNo3] THEN
             FollowerSeq(ExeCute:=TRUE , Next:= 130); 	
	     ELSE 
		     FollowerSeq(ExeCute:=TRUE , Next:= 200); //往皮带4倒药	
         END_IF
	130:  
	      ref_Follower.i.Pos:=ref_Follower.i.Pos+200;
	      FollowerSeq(ExeCute:=TRUE ,Hold:=FALSE, Next:= 150);
	
	150:
	      ref_Follower.i.MoveAbs:=TRUE;
		  IF ref_Follower.o.CmdDone THEN
			 ref_Follower.i.MoveAbs:=FALSE;
			 FollowerSeq(ExeCute:=TRUE ,Hold:=FALSE, Next:= 300);
		  END_IF
	
	//往皮带4落料
	200:
	     IF glb_BinBelt4_5.bin[1].arDrop[1] THEN
			FollowerSeq(ExeCute:=TRUE , Next:= 210); 
		 END_IF
		 IF Ref_MachineStateModel.Sts_Stopping  THEN
		    FollowerSeq(ExeCute:=TRUE , Next:= Seq_Stopping);   
	     END_IF
	
	210:
		ref_Follower.i.Pos:=ref_Follower.i.Pos+200;
		FollowerSeq(ExeCute:=TRUE ,Hold:=FALSE, Next:= 220);
	
	220:
	      ref_Follower.i.MoveAbs:=TRUE;
		  IF ref_Follower.o.CmdDone THEN
			 ref_Follower.i.MoveAbs:=FALSE;
			 FollowerSeq(ExeCute:=TRUE ,Hold:=FALSE, Next:= 230);
		  END_IF	
		  IF (ref_Follower.i.Pos-ref_Follower.o.ActPos) < 60 AND NOT bBeltInRange THEN
				glb_BinBelt4_5.bin[1].arDrop[1]:=FALSE;
				glb_BinBelt4_5.bin[1].Name:= glb_BinBelt3.bin[HMI_B3DropBinNo3].Name;
				glb_BinBelt4_5.bin[1].Amount:= glb_BinBelt3.bin[HMI_B3DropBinNo3].Amount;
				glb_BinBelt4_5.bin[1].bReject:= glb_BinBelt3.bin[HMI_B3DropBinNo3].bReject;
				glb_lrBelt3ValidCnt:=glb_lrBelt3ValidCnt-1;
			  bBeltInRange:=TRUE;
		  END_IF 
	
	230:  
	      bBeltInRange:=FALSE;
		  glb_BinBelt3.bin[HMI_B3DropBinNo3].arDrop[HMI_B3DropBinNo3]:=FALSE;
		  FollowerSeq(ExeCute:=TRUE ,Hold:=FALSE, Next:= 300); 
		  
    300: 
	
			FOR i:=64 TO 1 BY -1 DO
				glb_BinBelt3.bin[i]:= glb_BinBelt3.bin[i-1];  
			END_FOR	     
			glb_BinBelt3.bin[1].arDrop[HMI_B3DropBinNo1]:=FALSE;
			glb_BinBelt3.bin[1].arDrop[HMI_B3DropBinNo2]:=FALSE;
			glb_BinBelt3.bin[1].arDrop[HMI_B3DropBinNo3]:=FALSE;
			glb_lrBelt3WrkCnt:=glb_lrBelt3WrkCnt+1;
			FollowerSeq(ExeCute:=TRUE ,Hold:=FALSE, Next:= 111);  

			
		  
	Seq_Stopping: 
        iLastSeq:= FollowerSeq.Last; 
	    tonFollowerSeq(IN:=TRUE , PT:=T#1S , Q=> , ET=> );
		IF tonFollowerSeq.Q THEN
			tonFollowerSeq(IN:=FALSE , PT:=T#1S , Q=> , ET=> );
			FollowerSeq(ExeCute:=TRUE , Next:= Seq_StoppingDone); 
		END_IF
		
	Seq_StoppingDone:
	     ref_Follower.i.Disable:=TRUE;
		 IF NOT Ref_MachineStateModel.Sts_Stopping THEN
			FollowerSeq(ExeCute:=TRUE , Next:= 0); 
		 END_IF
END_CASE
FollowerSeq.Hold := Ref_MachineStateModel.Sts_Held;
END_ACTION

ACTION MainRoution:
EM_No:=4;
IF Ref_Unit.EM_Selected[EM_No] THEN
	IF Ref_MachineStateModel.Sts_Holding THEN
		Ref_Unit.EM_Holding_Done[EM_No]:=TRUE;
		ELSE
		Ref_Unit.EM_Holding_Done[EM_No]:=FALSE;
	END_IF
	IF Ref_MachineStateModel.Sts_UnHolding THEN
		Ref_Unit.EM_UnHolding_Done[EM_No]:=TRUE;
		ELSE
		Ref_Unit.EM_UnHolding_Done[EM_No]:=FALSE;
	END_IF
	
	IF Ref_MachineStateModel.Sts_Suspending THEN
		Ref_Unit.EM_Suspending_Done[EM_No]:=TRUE;
		ELSE
		Ref_Unit.EM_Suspending_Done[EM_No]:=FALSE;
	END_IF
	
	IF Ref_MachineStateModel.Sts_UnSuspending THEN
		Ref_Unit.EM_UnSuspending_Done[EM_No]:=TRUE;
		ELSE
		Ref_Unit.EM_UnSuspending_Done[EM_No]:=FALSE;
	END_IF
	
	IF Ref_MachineStateModel.Sts_Resetting AND FollowerSeq.Now=Seq_ResettingDone THEN
	   Ref_Unit.EM_Resetting_Done[EM_No]:=TRUE;
       ELSE   
	   Ref_Unit.EM_Resetting_Done[EM_No]:=FALSE;
	END_IF
	
	IF Ref_MachineStateModel.Sts_Clearing THEN
	   Ref_Unit.EM_Clearing_Done[EM_No]:=TRUE;
	   ELSE
	   Ref_Unit.EM_Clearing_Done[EM_No]:=FALSE;
	END_IF
	
	IF Ref_MachineStateModel.Sts_Starting THEN
	   Ref_Unit.EM_Starting_Done[EM_No]:=TRUE;
	   ELSE
       Ref_Unit.EM_Starting_Done[EM_No]:=FALSE;
	END_IF
	
	IF Ref_MachineStateModel.Sts_Stopping AND FollowerSeq.Now=Seq_StoppingDone  THEN
	   Ref_Unit.EM_Stopping_Done[EM_No]:=TRUE;	
       ELSE  
	   Ref_Unit.EM_Stopping_Done[EM_No]:=FALSE;	
	END_IF

	IF Ref_MachineStateModel.Sts_Aborting THEN
	    FollowerSeq(ExeCute:=TRUE , Next:= 0);	
		IF ref_Follower.o.InSync THEN	 
		   ref_Follower.i.CamOut:=TRUE;
		ELSE IF  NOT ref_Follower.o.StandStill THEN
				ref_follower.i.Stop:=TRUE;
			END_IF
		END_IF  
		
		IF tonAbortingWatchDog.Q THEN 
			Ref_Unit.EM_Aborting_Done[EM_No]:=TRUE;
			ref_Follower.i.Disable:=TRUE;
        END_IF
    ELSE
		Ref_Unit.EM_Aborting_Done[EM_No]:=FALSE;
	END_IF
	
	tonAbortingWatchDog(IN:= Ref_MachineStateModel.Sts_Aborting, PT:=T#3S , Q=> , ET=> );
	CM02_Follower();
ELSE
FollowerSeq(ExeCute:=TRUE , Next:= 0); 			
END_IF
END_ACTION

ACTION SR999_FaultHandler:
;
END_ACTION

END_PROGRAM

// ---- POUs/PackMaL_UN01/EM05_Counters.TcPOU
PROGRAM EM05_Counters
VAR
	ref_Master: REFERENCE TO UDT_AXISADMIN;
	Ref_MachineStateModel: REFERENCE TO PackMlv3_StateModel;
	Ref_Unit: REFERENCE TO UDT_UnitAdmin;	
	
	ref_Work_Recipe: REFERENCE TO UDT_Hmi_Output; //当前生产的配方反馈给触摸屏
	ref_diBeltObjCnt: REFERENCE TO DINT;
	ref_lrLatchMasterPos: REFERENCE TO LREAL;
    ref_lrMasterTargetPos: REFERENCE TO LREAL;
	ref_BinList: REFERENCE TO UDT_BINlist;
	
	EM_No: INT:=5;
	diProductCnt: DINT;
	tonAbortingWatchDog: TON;
	i,j,k: INT;

	rt_ProductCntUp: R_Trig;
	
	arDropFlag: ARRAY[1..40] OF BOOL;//落料标志	
	arDropCnt: ARRAY[1..40] OF DINT;//落料技数


	tonExeRtirg: ARRAY [1..40 ] OF Ton;
	arDropInRange: ARRAY [1..40 ] OF BOOL;
	d: INT;
	rtDropInRange: ARRAY [1..40 ] OF R_trig;
	ftDropFlag: ARRAY [1..40 ] OF F_trig;
	rtDropFlag: ARRAY [1..40 ] OF R_trig;
	ftInSensor: ARRAY [1..40 ] OF F_trig;
	rtInSensor: ARRAY [1..40 ] OF R_trig;
	ftOutSensor: ARRAY [1..40 ] OF F_trig;
	rtOutSensor: ARRAY [1..40 ] OF R_trig;	

	iNotDone: INT;

	iHomeCnt: INT;
	iPowerCnt: INT;
	iInitDone: INT;
	iStandstill: INT;
	Loc_Counter_Seq: INT;

	diMasterRangeCnt: DINT; //出料皮带计数
	aoi_binProduct: AOI_BIN;
	rtBeltInRange: R_trig;
	lrMasterPosAdd: LREAL;
	lrWorkPosBuffer: LREAL;
	iNotInitID: INT;

	iMovAbsCnt: INT;

	lrWorkPosExe: LREAL;
	iC: INT;
	iB: INT;
	iMovFailCnt: INT;
	
	
	tonCounterSeq: Ton;
	CounterSeq: SequenceTransfer;
	
	iDrop: INT;
	iBusyCounter: INT;
	iNotBusyCounter: INT;
	iCntDone: INT;
END_VAR

VAR CONSTANT
;
END_VAR

//伺服转1圈 落料24颗
Ref_MachineStateModel REF= UN01_MachineStateModel;
Ref_Unit REF=Unit01;
ref_Work_Recipe REF=HMI_Output;
ref_Master REF= arVirtualAxisAdmin[1];
ref_diBeltObjCnt REF=glb_diBeltObjCnt;

ref_BinList REF= Glb_BinList;
MainRoution();

ACTION CM01_Counters:
CASE CounterSeq.Now OF
	0: 
	   IF Ref_MachineStateModel.Sts_Resetting THEN
          CounterSeq(ExeCute:= TRUE, Next:= Seq_Resetting);
	   END_IF	
	   IF Ref_MachineStateModel.Sts_Stopping  THEN
          CounterSeq(ExeCute:= TRUE, Next:= Seq_Stopping);
	   END_IF
	   IF Ref_MachineStateModel.Sts_Execute  THEN
		  CounterSeq(ExeCute:= TRUE, Next:= 110);   
	   END_IF	 	   
	Seq_Resetting:
	  iPowerCnt:=0;
		FOR i:=1 TO 40 DO
			IF NOT arRealAxisAdmin[i].o.PowerOn THEN
			   arRealAxisAdmin[i].i.Enable:=TRUE;
			ELSE
			   iPowerCnt:=iPowerCnt+1;
			END_IF  
		END_FOR
		IF iPowerCnt=40 THEN
		   CounterSeq(ExeCute:= TRUE, Next:= 11);
		END_IF
		IF Ref_MachineStateModel.Sts_Stopping  THEN
		   CounterSeq(ExeCute:= TRUE, Next:= Seq_Stopping);
		END_IF	  
		
	11:
       tonCounterSeq(IN:=TRUE , PT:=T#1S , Q=> , ET=> );
	   IF tonCounterSeq.Q THEN
          tonCounterSeq(IN:=FALSE , PT:=T#1S , Q=> , ET=> );	
          CounterSeq(ExeCute:= TRUE, Next:= 20);
	   END_IF
	   
	20:
		IF NOT glb_AllAxisHomed_UN01 THEN
			CounterSeq(ExeCute:=TRUE , Next:= 21);  
			ELSE
			CounterSeq(ExeCute:=TRUE , Next:= 30); 
		END_IF	
	21:
	   iHomeCnt:=0;
	   FOR i:=1 TO 40 DO
		   arRealAxisAdmin[i].i.Pos:=0;
		   arRealAxisAdmin[i].i.HomeMode:=2;
		   arRealAxisAdmin[i].i.Home:=TRUE;    
		   IF arRealAxisAdmin[i].o.HomeDone THEN
			   iHomeCnt:=iHomeCnt+1;
		   END_IF     
	   END_FOR   
	   
	   IF iHomeCnt=40 THEN
          CounterSeq(ExeCute:= TRUE, Next:= 22);
	   END_IF	
       IF Ref_MachineStateModel.Sts_Stopping  THEN
	      CounterSeq(ExeCute:= TRUE, Next:= Seq_Stopping);
	   END_IF
		   
    22:
       tonCounterSeq(IN:=TRUE , PT:=T#1S , Q=> , ET=> );
	   IF tonCounterSeq.Q THEN
          tonCounterSeq(IN:=FALSE , PT:=T#1S , Q=> , ET=> );	
          CounterSeq(ExeCute:= TRUE, Next:= 23);
	   END_IF
          
	23:
       FOR  i:=1 TO 40 DO
		   arRealAxisAdmin[i].i.Home:=FALSE;
	   END_FOR

       CounterSeq(ExeCute:= TRUE, Next:= 30);
   
	30:
	    iNotBusyCounter:=0;
	    FOR i:=1 TO 40 DO
			IF NOT arCounters[i].Busy THEN
				iNotBusyCounter:=iNotBusyCounter+1;
			ELSE
				iBusyCounter:=i;
			END_IF	
		END_FOR
		IF iNotBusyCounter=40 THEN
           CounterSeq(ExeCute:= TRUE, Next:= 40);
	    ELSE IF Ref_MachineStateModel.Sts_Stopping  THEN
			    CounterSeq(ExeCute:= TRUE, Next:= Seq_Stopping);
			 END_IF	
		END_IF
		
    40:		
		tonCounterSeq(IN:=TRUE , PT:=T#1S , Q=> , ET=> );
		IF tonCounterSeq.Q THEN
		   tonCounterSeq(IN:=FALSE , PT:=T#1S , Q=> , ET=> );	
		   CounterSeq(ExeCute:= TRUE, Next:= Seq_ResettingDone);
		END_IF    

	Seq_ResettingDone:
		IF NOT Ref_MachineStateModel.Sts_Resetting THEN
		   CounterSeq(ExeCute:= TRUE, Next:= 0);
		END_IF	
	  
    110:
		   IF HMI_Output.RecipeModifyDone THEN
				FOR i:=1 TO 40 DO 
					arCounters[i].Enable:=TRUE;		
				END_FOR	
           ELSE
				FOR i:=1 TO 40 DO 
					arCounters[i].Enable:=FALSE;		
				END_FOR				   
		   END_IF
	
		
	   IF Ref_MachineStateModel.Sts_Stopping  THEN
          CounterSeq(ExeCute:= TRUE, Next:= Seq_Stopping);
	   END_IF		
		
		
		
		
	Seq_Stopping: 	
		iNotBusyCounter:=0;
		FOR i:=1 TO 40 DO
			IF NOT arCounters[i].Busy THEN
				iNotBusyCounter:=iNotBusyCounter+1;
			ELSE
				iBusyCounter:=i;
			END_IF	
		END_FOR
		IF iNotBusyCounter=40 THEN
		   CounterSeq(ExeCute:= TRUE, Next:= 903);
		END_IF
	
	
	903:
		FOR i:=1 TO 40 DO 
			arCounters[i].Enable:=FALSE;	
            arCounters[i].Execute:=FALSE;	
            CounterSeq(ExeCute:= TRUE, Next:= 904);	
		END_FOR	
    904:
		tonCounterSeq(IN:=TRUE , PT:=T#1.5S , Q=> , ET=> );	  
		IF tonCounterSeq.Q THEN
			tonCounterSeq(IN:=FALSE , PT:=T#1.5S , Q=> , ET=> );	
			CounterSeq(ExeCute:= TRUE, Next:= 905);  
		END_IF				

	905:
	    FOR i:=1 TO 40 DO 
			arRealAxisAdmin[i].i.Disable:=TRUE;
			CounterSeq(ExeCute:= TRUE, Next:= Seq_StoppingDone);
        END_FOR	
			
	
	Seq_StoppingDone:
		IF NOT Ref_MachineStateModel.Sts_Stopping THEN
		   CounterSeq(ExeCute:= TRUE, Next:= 0);
		END_IF	
		
END_CASE
END_ACTION

ACTION MainRoution:
EM_No:=5;
IF Ref_Unit.EM_Selected[EM_No] THEN
	IF Ref_MachineStateModel.Sts_Holding THEN
		Ref_Unit.EM_Holding_Done[EM_No]:=TRUE;
		ELSE
		Ref_Unit.EM_Holding_Done[EM_No]:=FALSE;
	END_IF
	IF Ref_MachineStateModel.Sts_UnHolding THEN
		Ref_Unit.EM_UnHolding_Done[EM_No]:=TRUE;
		ELSE
		Ref_Unit.EM_UnHolding_Done[EM_No]:=FALSE;
	END_IF
	
	IF Ref_MachineStateModel.Sts_Suspending THEN
		Ref_Unit.EM_Suspending_Done[EM_No]:=TRUE;
		ELSE
		Ref_Unit.EM_Suspending_Done[EM_No]:=FALSE;
	END_IF
	
	IF Ref_MachineStateModel.Sts_UnSuspending THEN
		Ref_Unit.EM_UnSuspending_Done[EM_No]:=TRUE;
		ELSE
		Ref_Unit.EM_UnSuspending_Done[EM_No]:=FALSE;
	END_IF
	
	IF Ref_MachineStateModel.Sts_Resetting AND CounterSeq.Now=Seq_ResettingDone THEN
       Ref_Unit.EM_Resetting_Done[EM_No]:=TRUE;
       ELSE   
       Ref_Unit.EM_Resetting_Done[EM_No]:=FALSE;	   
	END_IF
	
	IF Ref_MachineStateModel.Sts_Clearing THEN
	   Ref_Unit.EM_Clearing_Done[EM_No]:=TRUE;
	   ELSE   
	   Ref_Unit.EM_Clearing_Done[EM_No]:=FALSE;
	END_IF
	
	IF Ref_MachineStateModel.Sts_Starting THEN
	   Ref_Unit.EM_Starting_Done[EM_No]:=TRUE;
	   ELSE	   
	   Ref_Unit.EM_Starting_Done[EM_No]:=FALSE;
	END_IF
	
	IF Ref_MachineStateModel.Sts_Stopping AND CounterSeq.Now=Seq_StoppingDone THEN
	   Ref_Unit.EM_Stopping_Done[EM_No]:=TRUE;	
	   ELSE
	   Ref_Unit.EM_Stopping_Done[EM_No]:=FALSE;	   
	END_IF

	IF Ref_MachineStateModel.Sts_Aborting THEN
		CounterSeq(ExeCute:= TRUE, Next:= 0);
        FOR i:=1 TO 40 DO 
			arCounters[i].Enable:=FALSE; 
			arDropCylinder[i].i.ActiveIn:=FALSE;
			arDropCylinder[i].i.ActiveOut:=FALSE;
		END_FOR
		
		IF  tonAbortingWatchDog.Q THEN 
		    Ref_Unit.EM_Aborting_Done[EM_No]:=TRUE;
			FOR i:=1 TO 40 DO 
				arRealAxisAdmin[i].i.Enable:=FALSE;
			END_FOR			
		END_IF
		ELSE
        Ref_Unit.EM_Aborting_Done[EM_No]:=FALSE;
	END_IF
	tonAbortingWatchDog(IN:= Ref_MachineStateModel.Sts_Aborting, PT:=T#3S , Q=> , ET=> );	
CM01_Counters();
ELSE
	CounterSeq(ExeCute:= TRUE, Next:= 0);
END_IF
END_ACTION

ACTION SR999_FaultHandler:
;
END_ACTION

END_PROGRAM

// ---- Add-On-Instructions/AOI_Bin.TcPOU
FUNCTION_BLOCK AOI_Bin
VAR_INPUT
	Trigger: BOOL;
	BeltPos: LREAL;
	PosOffset: LREAL;
	RangeValue: LREAL:=10;
	Valid: BOOL;
END_VAR
VAR_OUTPUT
END_VAR
VAR
	rtTrig: R_trig;
	i: USINT;
	j: INT;
	k: USINT;
	arPosDiff: array[0..254] of LREAL;
	lrPosDiff1: LREAL;
	diInRangCnt: DINT;
	h: INT;
END_VAR
VAR_IN_OUT
	BinList: UDT_BinList;
END_VAR

rtTrig(CLK:=Trigger , Q=> );

IF rtTrig.Q THEN
	BinList.Bin[0].lrlatchPos:=BeltPos;	
    BinList.Bin[0].bValid:=Valid;
  	FOR k:=254 TO 1 BY -1 DO
		BinList.Bin[k].bValid:=binlist.Bin[k-1].bValid;
		BinList.Bin[k].bReject:=binlist.Bin[k-1].bReject;
		BinList.Bin[k].lrlatchPos:=binlist.Bin[k-1].lrlatchPos;
	END_FOR
    BinList.Bin[0].bValid:= FALSE;
    BinList.Bin[0].bReject:= FALSE;	
END_IF


FOR i:=128 TO 1 BY -1 DO
    IF BinList.Bin[i].bValid THEN
       arPosDiff[i]:= BeltPos-BinList.bin[i].lrlatchPos;	
  	END_IF
END_FOR

FOR j:=1 TO 20 DO
   diInRangCnt:=0;
   FOR i:=128 TO 1 BY -1 DO
		IF arPosDiff[i]> BinList.arWorkPos[j] + PosOffset
		AND arPosDiff[i] < (BinList.arWorkPos[j]+PosOffset+ RangeValue) THEN
			diInRangCnt:=diInRangCnt+1;
		END_IF 
   END_FOR
   IF diInRangCnt<>0 THEN
	  BinList.arInRang[j]:=TRUE; 
	  ELSE
	  BinList.arInRang[j]:=FALSE;
   END_IF
   
END_FOR



IF BinList.Reset THEN
	FOR h:=0 TO 254  DO
		BinList.Bin[h].bValid:=FALSE;
		BinList.Bin[h].bReject:=FALSE;
	END_FOR
END_IF

END_FUNCTION_BLOCK

// ---- POUs/PackMaL_UN01/EM06_Follower4_5.TcPOU
PROGRAM EM06_Follower4_5
VAR
	ref_Master: REFERENCE TO UDT_AXISADMIN;
	ref_Follower1: REFERENCE TO UDT_AXISADMIN;
	ref_Follower2: REFERENCE TO UDT_AXISADMIN;
	Ref_MachineStateModel: REFERENCE TO PackMlv3_StateModel;
	Ref_Unit: REFERENCE TO UDT_UnitAdmin;	
	Loc_Resetting_Seq: INT;//
	EM_No: INT:=6;
	tonAbortingWatchDog: TON;

	
	MC_GearIn_Follower1: MC_GearIn;
	MC_CamIn_Follower1: MC_CamIn_V2;
	MC_CamTableSelect_Follower1: MC_CamTableSelect;
	CamTableFollower1: MC_CAM_REF;
	MC_GearIn_Follower2: MC_GearIn;
	MC_CamIn_Follower2: MC_CamIn_v2;
	MC_CamTableSelect_Follower2: MC_CamTableSelect;
	CamTableFollower2: MC_CAM_REF;
	
    MC_ReadCamTableSlaveDynamicsFollwer1: MC_ReadCamTableSlaveDynamics;
    MC_ReadCamTableSlaveDynamicsFollwer2: MC_ReadCamTableSlaveDynamics;
	
	table1: ARRAY[1..255] OF MC_MotionFunctionPoint; (*用于定义电子凸轮表中的关键点*)
	table2: ARRAY[1..255] OF MC_MotionFunctionPoint; (*用于定义电子凸轮表中的关键点*)

	lrFollower2PosLast: LREAL;
	diPos1Mod: DINT;
	diPos2Mod: DINT;
	rtInDropPos: r_trig;


	iInDropPosCnt: INT;
	tonFollowerSeqDelay: Ton;
	lrFollow1CamDynPos: LREAL;
	lrFollow2CamDynPos: LREAL;
	lrFollow2LatchPos: LREAL;
	lrFollow1LatchPos: LREAL;


